LIN {X 0,Y 188.353,Z 512.177,A -85,B 0,C 180,E1 -22070.571,E2 -22070.571} C_VEL
LIN {X 0,Y 190.669,Z 502.352,A -85,B 0,C 180,E1 -22073.346,E2 -22073.346} C_VEL
LIN {X 0,Y 192.539,Z 493.281,A -85,B 0,C 180,E1 -22075.401,E2 -22075.401} C_VEL
LIN {X 0,Y 194.201,Z 485.139,A -85,B 0,C 180,E1 -22076.899,E2 -22076.899} C_VEL
LIN {X 0,Y 196.354,Z 473.565,A -85,B 0,C 180,E1 -22078.605,E2 -22078.605} C_VEL
LIN {X 0,Y 198.216,Z 461.568,A -85,B 0,C 180,E1 -22079.911,E2 -22079.911} C_VEL
LIN {X 0,Y 199.572,Z 449.492,A -85,B 0,C 180,E1 -22080.855,E2 -22080.855} C_VEL
LIN {X 0,Y 200.443,Z 436.398,A -85,B 0,C 180,E1 -22081.513,E2 -22081.513} C_VEL
LIN {X 0,Y 202.303,Z 391.383,A -85,B 0,C 180,E1 -22083.04,E2 -22083.04} C_VEL
LIN {X 0,Y 199.367,Z 363.798,A -85,B 0,C 180,E1 -22084.587,E2 -22084.587} C_VEL
LIN {X 0,Y 192.816,Z 346.528,A -85,B 0,C 180,E1 -22086.384,E2 -22086.384} C_VEL
LIN {X 0,Y 187.657,Z 334.98,A -85,B 0,C 180,E1 -22087.815,E2 -22087.815} C_VEL
LIN {X 0,Y 186.775,Z 332.616,A -85,B 0,C 180,E1 -22088.175,E2 -22088.175} C_VEL
LIN {X 0,Y 185.486,Z 327.382,A -85,B 0,C 180,E1 -22091.001,E2 -22091.001} C_VEL
LIN {X 0,Y 185.466,Z 327.381,A -85,B 0,C 180,E1 -22096.057,E2 -22096.057} C_VEL
LIN {X 0,Y 185.475,Z 327.377,A -85,B 0,C 180,E1 -22099.896,E2 -22099.896} C_VEL
LIN {X 0,Y 185.514,Z 327.371,A -85,B 0,C 180,E1 -22102.713,E2 -22102.713} C_VEL
LIN {X 0,Y 185.555,Z 327.368,A -85,B 0,C 180,E1 -22107.977,E2 -22107.977} C_VEL
LIN {X 0,Y 185.591,Z 327.36,A -85,B 0,C 180,E1 -22110.577,E2 -22110.577} C_VEL
LIN {X 0,Y 185.589,Z 327.367,A -85,B 0,C 180,E1 -22115.382,E2 -22115.382} C_VEL
LIN {X 0,Y 185.552,Z 327.357,A -85,B 0,C 180,E1 -22120.069,E2 -22120.069} C_VEL
LIN {X 0,Y 185.678,Z 327.348,A -85,B 0,C 180,E1 -22124.635,E2 -22124.635} C_VEL
LIN {X 0,Y 185.897,Z 327.323,A -85,B 0,C 180,E1 -22129.419,E2 -22129.419} C_VEL
LIN {X 0,Y 185.944,Z 327.291,A -85,B 0,C 180,E1 -22133.489,E2 -22133.489} C_VEL
LIN {X 0,Y 186.21,Z 327.284,A -85,B 0,C 180,E1 -22137.837,E2 -22137.837} C_VEL
LIN {X 0,Y 186.412,Z 327.264,A -85,B 0,C 180,E1 -22140,E2 -22140} C_VEL
LIN {X 0,Y 185.922,Z 327.297,A -85,B 0,C 180,E1 -22144.335,E2 -22144.335} C_VEL
LIN {X 0,Y 185.989,Z 327.3,A -85,B 0,C 180,E1 -22148.693,E2 -22148.693} C_VEL
LIN {X 0,Y 185.727,Z 327.348,A -85,B 0,C 180,E1 -22153.123,E2 -22153.123} C_VEL
LIN {X 0,Y 185.664,Z 327.355,A -85,B 0,C 180,E1 -22157.627,E2 -22157.627} C_VEL
LIN {X 0,Y 185.581,Z 327.36,A -85,B 0,C 180,E1 -22162.253,E2 -22162.253} C_VEL
LIN {X 0,Y 185.568,Z 327.366,A -85,B 0,C 180,E1 -22167.031,E2 -22167.031} C_VEL
LIN {X 0,Y 185.586,Z 327.36,A -85,B 0,C 180,E1 -22169.491,E2 -22169.491} C_VEL
LIN {X 0,Y 185.506,Z 327.367,A -85,B 0,C 180,E1 -22174.63,E2 -22174.63} C_VEL
LIN {X 0,Y 185.513,Z 327.374,A -85,B 0,C 180,E1 -22177.311,E2 -22177.311} C_VEL
LIN {X 0,Y 185.477,Z 327.37,A -85,B 0,C 180,E1 -22180.723,E2 -22180.723} C_VEL
LIN {X 0,Y 185.464,Z 327.376,A -85,B 0,C 180,E1 -22186.053,E2 -22186.053} C_VEL
LIN {X 0,Y 185.472,Z 327.376,A -85,B 0,C 180,E1 -22189.893,E2 -22189.893} C_VEL
LIN {X 0,Y 185.511,Z 327.376,A -85,B 0,C 180,E1 -22192.709,E2 -22192.709} C_VEL
LIN {X 0,Y 185.546,Z 327.37,A -85,B 0,C 180,E1 -22197.972,E2 -22197.972} C_VEL
LIN {X 0,Y 185.585,Z 327.368,A -85,B 0,C 180,E1 -22200.574,E2 -22200.574} C_VEL
LIN {X 0,Y 185.68,Z 327.355,A -85,B 0,C 180,E1 -22206.578,E2 -22206.578} C_VEL
LIN {X 0,Y 185.67,Z 327.485,A -85,B 0,C 180,E1 -22207.071,E2 -22207.071} C_VEL
LIN {X 0,Y 186.702,Z 330.28,A -85,B 0,C 180,E1 -22207.396,E2 -22207.396} C_VEL
LIN {X 0,Y 194.168,Z 343.936,A -85,B 0,C 180,E1 -22209.343,E2 -22209.343} C_VEL
LIN {X 0,Y 200.218,Z 357.134,A -85,B 0,C 180,E1 -22210.88,E2 -22210.88} C_VEL
LIN {X 0,Y 203.246,Z 366.009,A -85,B 0,C 180,E1 -22211.697,E2 -22211.697} C_VEL
LIN {X 0,Y 200.358,Z 428.689,A -85,B 0,C 180,E1 -22213.831,E2 -22213.831} C_VEL
LIN {X 0,Y 199.181,Z 442.535,A -85,B 0,C 180,E1 -22214.717,E2 -22214.717} C_VEL
LIN {X 0,Y 197.731,Z 455.437,A -85,B 0,C 180,E1 -22215.984,E2 -22215.984} C_VEL
LIN {X 0,Y 195.76,Z 467.279,A -85,B 0,C 180,E1 -22217.558,E2 -22217.558} C_VEL
LIN {X 0,Y 193.815,Z 478.594,A -85,B 0,C 180,E1 -22219.551,E2 -22219.551} C_VEL
LIN {X 0,Y 191.557,Z 488.867,A -85,B 0,C 180,E1 -22221.824,E2 -22221.824} C_VEL
LIN {X 0,Y 189.243,Z 498.9,A -85,B 0,C 180,E1 -22224.67,E2 -22224.67} C_VEL
LIN {X 0,Y 187.126,Z 507.738,A -85,B 0,C 180,E1 -22227.844,E2 -22227.844} C_VEL
LIN {X 0,Y 185.539,Z 514.774,A -85,B 0,C 180,E1 -22231.082,E2 -22231.082} C_VEL
LIN {X 0,Y 184.434,Z 520.402,A -85,B 0,C 180,E1 -22234.368,E2 -22234.368} C_VEL
LIN {X 0,Y 183.638,Z 524.836,A -85,B 0,C 180,E1 -22237.694,E2 -22237.694} C_VEL
LIN {X 0,Y 183.048,Z 528.196,A -85,B 0,C 180,E1 -22241.064,E2 -22241.064} C_VEL
LIN {X 0,Y 182.893,Z 529.868,A -85,B 0,C 180,E1 -22243.327,E2 -22243.327} C_VEL
LIN {X 0,Y 182.926,Z 531.341,A -85,B 0,C 180,E1 -22246.159,E2 -22246.159} C_VEL
LIN {X 0,Y 183.339,Z 532.303,A -85,B 0,C 180,E1 -22250.178,E2 -22250.178} C_VEL
LIN {X 0,Y 184.263,Z 532.066,A -85,B 0,C 180,E1 -22253.741,E2 -22253.741} C_VEL
LIN {X 0,Y 185.539,Z 530.916,A -85,B 0,C 180,E1 -22257.032,E2 -22257.032} C_VEL
LIN {X 0,Y 187.356,Z 528.771,A -85,B 0,C 180,E1 -22260.373,E2 -22260.373} C_VEL
LIN {X 0,Y 189.807,Z 525.491,A -85,B 0,C 180,E1 -22263.734,E2 -22263.734} C_VEL
LIN {X 0,Y 192.877,Z 520.967,A -85,B 0,C 180,E1 -22267.041,E2 -22267.041} C_VEL
LIN {X 0,Y 196.347,Z 515.364,A -85,B 0,C 180,E1 -22270.108,E2 -22270.108} C_VEL
LIN {X 0,Y 200.451,Z 508.123,A -85,B 0,C 180,E1 -22273.128,E2 -22273.128} C_VEL
LIN {X 0,Y 204.18,Z 500.616,A -85,B 0,C 180,E1 -22275.575,E2 -22275.575} C_VEL
LIN {X 0,Y 208.336,Z 491.441,A -85,B 0,C 180,E1 -22277.91,E2 -22277.91} C_VEL
LIN {X 0,Y 212.331,Z 481.267,A -85,B 0,C 180,E1 -22279.939,E2 -22279.939} C_VEL
LIN {X 0,Y 215.607,Z 471.5,A -85,B 0,C 180,E1 -22281.467,E2 -22281.467} C_VEL
LIN {X 0,Y 218.521,Z 460.893,A -85,B 0,C 180,E1 -22282.785,E2 -22282.785} C_VEL
LIN {X 0,Y 221.185,Z 448.606,A -85,B 0,C 180,E1 -22283.921,E2 -22283.921} C_VEL
LIN {X 0,Y 223.29,Z 435.152,A -85,B 0,C 180,E1 -22284.784,E2 -22284.784} C_VEL
LIN {X 0,Y 224.598,Z 421.235,A -85,B 0,C 180,E1 -22285.305,E2 -22285.305} C_VEL
LIN {X 0,Y 226.623,Z 388.171,A -85,B 0,C 180,E1 -22286.294,E2 -22286.294} C_VEL
LIN {X 0,Y 221.369,Z 377.129,A -85,B 0,C 180,E1 -22288.355,E2 -22288.355} C_VEL
LIN {X 0,Y 217.126,Z 369.65,A -85,B 0,C 180,E1 -22290.088,E2 -22290.088} C_VEL
LIN {X 0,Y 211.412,Z 360.897,A -85,B 0,C 180,E1 -22292.6,E2 -22292.6} C_VEL
LIN {X 0,Y 205.592,Z 352.678,A -85,B 0,C 180,E1 -22295.44,E2 -22295.44} C_VEL
LIN {X 0,Y 202.329,Z 348.373,A -85,B 0,C 180,E1 -22297.188,E2 -22297.188} C_VEL
LIN {X 0,Y 199.485,Z 344.709,A -85,B 0,C 180,E1 -22298.832,E2 -22298.832} C_VEL
LIN {X 0,Y 198.733,Z 343.71,A -85,B 0,C 180,E1 -22299.29,E2 -22299.29} C_VEL
LIN {X 0,Y 196.069,Z 340.766,A -85,B 0,C 180,E1 -22300.977,E2 -22300.977} C_VEL
LIN {X 0,Y 194.761,Z 338.596,A -85,B 0,C 180,E1 -22301.92,E2 -22301.92} C_VEL
LIN {X 0,Y 192.179,Z 336.315,A -85,B 0,C 180,E1 -22303.741,E2 -22303.741} C_VEL
LIN {X 0,Y 190.522,Z 333.195,A -85,B 0,C 180,E1 -22305.173,E2 -22305.173} C_VEL
LIN {X 0,Y 187.93,Z 331.617,A -85,B 0,C 180,E1 -22307.309,E2 -22307.309} C_VEL
LIN {X 0,Y 186.403,Z 329.386,A -85,B 0,C 180,E1 -22308.859,E2 -22308.859} C_VEL
LIN {X 0,Y 185.903,Z 327.319,A -85,B 0,C 180,E1 -22309.598,E2 -22309.598} C_VEL
LIN {X 0,Y 185.927,Z 327.307,A -85,B 0,C 180,E1 -22313.489,E2 -22313.489} C_VEL
LIN {X 0,Y 186.192,Z 327.272,A -85,B 0,C 180,E1 -22317.837,E2 -22317.837} C_VEL
LIN {X 0,Y 186.394,Z 327.258,A -85,B 0,C 180,E1 -22320,E2 -22320} C_VEL
LIN {X 0,Y 185.911,Z 327.309,A -85,B 0,C 180,E1 -22324.337,E2 -22324.337} C_VEL
LIN {X 0,Y 185.997,Z 327.295,A -85,B 0,C 180,E1 -22328.694,E2 -22328.694} C_VEL
LIN {X 0,Y 185.753,Z 327.328,A -85,B 0,C 180,E1 -22333.122,E2 -22333.122} C_VEL
LIN {X 0,Y 185.679,Z 327.343,A -85,B 0,C 180,E1 -22337.626,E2 -22337.626} C_VEL
LIN {X 0,Y 185.633,Z 327.508,A -85,B 0,C 180,E1 -22343.129,E2 -22343.129} C_VEL
LIN {X 0,Y 186.049,Z 329.192,A -85,B 0,C 180,E1 -22345.335,E2 -22345.335} C_VEL
LIN {X 0,Y 187.524,Z 331.42,A -85,B 0,C 180,E1 -22346.878,E2 -22346.878} C_VEL
LIN {X 0,Y 191.885,Z 336.607,A -85,B 0,C 180,E1 -22350.627,E2 -22350.627} C_VEL
LIN {X 0,Y 195.187,Z 341.306,A -85,B 0,C 180,E1 -22353.094,E2 -22353.094} C_VEL
LIN {X 0,Y 197.203,Z 343.952,A -85,B 0,C 180,E1 -22354.446,E2 -22354.446} C_VEL
LIN {X 0,Y 200.298,Z 348.364,A -85,B 0,C 180,E1 -22356.375,E2 -22356.375} C_VEL
LIN {X 0,Y 205.123,Z 355.887,A -85,B 0,C 180,E1 -22359.103,E2 -22359.103} C_VEL
LIN {X 0,Y 209.046,Z 362.3,A -85,B 0,C 180,E1 -22361.114,E2 -22361.114} C_VEL
LIN {X 0,Y 213.437,Z 369.913,A -85,B 0,C 180,E1 -22363.193,E2 -22363.193} C_VEL
LIN {X 0,Y 219.34,Z 381.612,A -85,B 0,C 180,E1 -22365.781,E2 -22365.781} C_VEL
LIN {X 0,Y 224.902,Z 394.525,A -85,B 0,C 180,E1 -22368.063,E2 -22368.063} C_VEL
LIN {X 0,Y 225.82,Z 397.48,A -85,B 0,C 180,E1 -22368.458,E2 -22368.458} C_VEL
LIN {X 0,Y 225.93,Z 401.219,A -85,B 0,C 180,E1 -22368.663,E2 -22368.663} C_VEL
LIN {X 0,Y 223.2,Z 441.55,A -85,B 0,C 180,E1 -22369.875,E2 -22369.875} C_VEL
LIN {X 0,Y 222.275,Z 449.228,A -85,B 0,C 180,E1 -22370.238,E2 -22370.238} C_VEL
LIN {X 0,Y 220.943,Z 454.939,A -85,B 0,C 180,E1 -22370.446,E2 -22370.446} C_VEL
LIN {X 0,Y 217.108,Z 464.094,A -85,B 0,C 180,E1 -22370.568,E2 -22370.568} C_VEL
LIN {X 0,Y 212.771,Z 472.95,A -85,B 0,C 180,E1 -22370.849,E2 -22370.849} C_VEL
LIN {X 0,Y 210.664,Z 478.188,A -85,B 0,C 180,E1 -22371.317,E2 -22371.317} C_VEL
LIN {X 0,Y 206.77,Z 489.566,A -85,B 0,C 180,E1 -22372.897,E2 -22372.897} C_VEL
LIN {X 0,Y 202.532,Z 499.986,A -85,B 0,C 180,E1 -22374.771,E2 -22374.771} C_VEL
LIN {X 0,Y 198.603,Z 508.522,A -85,B 0,C 180,E1 -22376.74,E2 -22376.74} C_VEL
LIN {X 0,Y 194.585,Z 516.413,A -85,B 0,C 180,E1 -22379.028,E2 -22379.028} C_VEL
LIN {X 0,Y 190.119,Z 524.183,A -85,B 0,C 180,E1 -22381.884,E2 -22381.884} C_VEL
LIN {X 0,Y 186.84,Z 529.738,A -85,B 0,C 180,E1 -22384.525,E2 -22384.525} C_VEL
LIN {X 0,Y 183.808,Z 534.686,A -85,B 0,C 180,E1 -22387.524,E2 -22387.524} C_VEL
LIN {X 0,Y 181.041,Z 538.753,A -85,B 0,C 180,E1 -22390.737,E2 -22390.737} C_VEL
LIN {X 0,Y 178.81,Z 541.797,A -85,B 0,C 180,E1 -22394.034,E2 -22394.034} C_VEL
LIN {X 0,Y 177.805,Z 543.321,A -85,B 0,C 180,E1 -22396.285,E2 -22396.285} C_VEL
LIN {X 0,Y 176.473,Z 545.123,A -85,B 0,C 180,E1 -22400.837,E2 -22400.837} C_VEL
LIN {X 0,Y 176.067,Z 545.411,A -85,B 0,C 180,E1 -22405.425,E2 -22405.425} C_VEL
LIN {X 0,Y 176.085,Z 544.94,A -85,B 0,C 180,E1 -22407.716,E2 -22407.716} C_VEL
LIN {X 0,Y 176.261,Z 544.069,A -85,B 0,C 180,E1 -22410.003,E2 -22410.003} C_VEL
LIN {X 0,Y 176.076,Z 541.728,A -85,B 0,C 180,E1 -22413.736,E2 -22413.736} C_VEL
LIN {X 0,Y 176.333,Z 537.6,A -85,B 0,C 180,E1 -22418.022,E2 -22418.022} C_VEL
LIN {X 0,Y 176.907,Z 533.014,A -85,B 0,C 180,E1 -22421.46,E2 -22421.46} C_VEL
LIN {X 0,Y 178.167,Z 526.023,A -85,B 0,C 180,E1 -22425.445,E2 -22425.445} C_VEL
LIN {X 0,Y 179.915,Z 518.437,A -85,B 0,C 180,E1 -22428.803,E2 -22428.803} C_VEL
LIN {X 0,Y 181.517,Z 511.685,A -85,B 0,C 180,E1 -22431.22,E2 -22431.22} C_VEL
LIN {X 0,Y 183.88,Z 502.268,A -85,B 0,C 180,E1 -22433.963,E2 -22433.963} C_VEL
LIN {X 0,Y 185.826,Z 493.232,A -85,B 0,C 180,E1 -22436.085,E2 -22436.085} C_VEL
LIN {X 0,Y 187.546,Z 485.126,A -85,B 0,C 180,E1 -22437.632,E2 -22437.632} C_VEL
LIN {X 0,Y 189.781,Z 473.623,A -85,B 0,C 180,E1 -22439.388,E2 -22439.388} C_VEL
LIN {X 0,Y 191.699,Z 461.749,A -85,B 0,C 180,E1 -22440.732,E2 -22440.732} C_VEL
LIN {X 0,Y 193.103,Z 449.847,A -85,B 0,C 180,E1 -22441.702,E2 -22441.702} C_VEL
LIN {X 0,Y 194.026,Z 437.151,A -85,B 0,C 180,E1 -22442.375,E2 -22442.375} C_VEL
LIN {X 0,Y 195.946,Z 391.813,A -85,B 0,C 180,E1 -22443.966,E2 -22443.966} C_VEL
LIN {X 0,Y 193.252,Z 365.907,A -85,B 0,C 180,E1 -22445.482,E2 -22445.482} C_VEL
LIN {X 0,Y 186.381,Z 347.697,A -85,B 0,C 180,E1 -22447.487,E2 -22447.487} C_VEL
LIN {X 0,Y 180.679,Z 335.314,A -85,B 0,C 180,E1 -22449.163,E2 -22449.163} C_VEL
LIN {X 0,Y 179.434,Z 332.329,A -85,B 0,C 180,E1 -22449.641,E2 -22449.641} C_VEL
LIN {X 0,Y 178.418,Z 328.26,A -85,B 0,C 180,E1 -22452.043,E2 -22452.043} C_VEL
LIN {X 0,Y 178.401,Z 328.264,A -85,B 0,C 180,E1 -22455.166,E2 -22455.166} C_VEL
LIN {X 0,Y 178.41,Z 328.26,A -85,B 0,C 180,E1 -22458.461,E2 -22458.461} C_VEL
LIN {X 0,Y 178.431,Z 328.255,A -85,B 0,C 180,E1 -22463.784,E2 -22463.784} C_VEL
LIN {X 0,Y 178.496,Z 328.244,A -85,B 0,C 180,E1 -22466.548,E2 -22466.548} C_VEL
LIN {X 0,Y 178.532,Z 328.238,A -85,B 0,C 180,E1 -22470.007,E2 -22470.007} C_VEL
LIN {X 0,Y 178.529,Z 328.247,A -85,B 0,C 180,E1 -22474.887,E2 -22474.887} C_VEL
LIN {X 0,Y 178.565,Z 328.219,A -85,B 0,C 180,E1 -22480.847,E2 -22480.847} C_VEL
LIN {X 0,Y 178.654,Z 328.229,A -85,B 0,C 180,E1 -22486.347,E2 -22486.347} C_VEL
LIN {X 0,Y 178.913,Z 328.181,A -85,B 0,C 180,E1 -22490.959,E2 -22490.959} C_VEL
LIN {X 0,Y 179.156,Z 328.162,A -85,B 0,C 180,E1 -22497.751,E2 -22497.751} C_VEL
LIN {X 0,Y 179.375,Z 328.14,A -85,B 0,C 180,E1 -22500,E2 -22500} C_VEL
LIN {X 0,Y 178.869,Z 328.173,A -85,B 0,C 180,E1 -22504.507,E2 -22504.507} C_VEL
LIN {X 0,Y 178.918,Z 328.183,A -85,B 0,C 180,E1 -22509.039,E2 -22509.039} C_VEL
LIN {X 0,Y 178.653,Z 328.228,A -85,B 0,C 180,E1 -22513.652,E2 -22513.652} C_VEL
LIN {X 0,Y 178.598,Z 328.238,A -85,B 0,C 180,E1 -22519.184,E2 -22519.184} C_VEL
LIN {X 0,Y 178.528,Z 328.247,A -85,B 0,C 180,E1 -22525.113,E2 -22525.113} C_VEL
LIN {X 0,Y 178.53,Z 328.24,A -85,B 0,C 180,E1 -22529.992,E2 -22529.992} C_VEL
LIN {X 0,Y 178.492,Z 328.242,A -85,B 0,C 180,E1 -22534.217,E2 -22534.217} C_VEL
LIN {X 0,Y 178.402,Z 328.256,A -85,B 0,C 180,E1 -22539.072,E2 -22539.072} C_VEL
LIN {X 0,Y 178.404,Z 328.258,A -85,B 0,C 180,E1 -22542.043,E2 -22542.043} C_VEL
LIN {X 0,Y 178.399,Z 328.255,A -85,B 0,C 180,E1 -22545.162,E2 -22545.162} C_VEL
LIN {X 0,Y 178.408,Z 328.259,A -85,B 0,C 180,E1 -22548.457,E2 -22548.457} C_VEL
LIN {X 0,Y 178.427,Z 328.256,A -85,B 0,C 180,E1 -22553.781,E2 -22553.781} C_VEL
LIN {X 0,Y 178.49,Z 328.252,A -85,B 0,C 180,E1 -22556.544,E2 -22556.544} C_VEL
LIN {X 0,Y 178.526,Z 328.248,A -85,B 0,C 180,E1 -22560.004,E2 -22560.004} C_VEL
LIN {X 0,Y 178.594,Z 328.324,A -85,B 0,C 180,E1 -22565.674,E2 -22565.674} C_VEL
LIN {X 0,Y 179.692,Z 331.231,A -85,B 0,C 180,E1 -22566.044,E2 -22566.044} C_VEL
LIN {X 0,Y 180.979,Z 333.249,A -85,B 0,C 180,E1 -22566.404,E2 -22566.404} C_VEL
LIN {X 0,Y 189.443,Z 349.04,A -85,B 0,C 180,E1 -22568.736,E2 -22568.736} C_VEL
LIN {X 0,Y 194.932,Z 361.55,A -85,B 0,C 180,E1 -22570.217,E2 -22570.217} C_VEL
LIN {X 0,Y 196.911,Z 367.636,A -85,B 0,C 180,E1 -22570.79,E2 -22570.79} C_VEL
LIN {X 0,Y 193.961,Z 429.467,A -85,B 0,C 180,E1 -22572.966,E2 -22572.966} C_VEL
LIN {X 0,Y 192.748,Z 442.893,A -85,B 0,C 180,E1 -22573.855,E2 -22573.855} C_VEL
LIN {X 0,Y 191.305,Z 455.251,A -85,B 0,C 180,E1 -22575.095,E2 -22575.095} C_VEL
LIN {X 0,Y 189.392,Z 466.403,A -85,B 0,C 180,E1 -22576.586,E2 -22576.586} C_VEL
LIN {X 0,Y 187.311,Z 477.935,A -85,B 0,C 180,E1 -22578.636,E2 -22578.636} C_VEL
LIN {X 0,Y 185.047,Z 488.117,A -85,B 0,C 180,E1 -22580.917,E2 -22580.917} C_VEL
LIN {X 0,Y 182.954,Z 496.91,A -85,B 0,C 180,E1 -22583.379,E2 -22583.379} C_VEL
LIN {X 0,Y 180.629,Z 506.146,A -85,B 0,C 180,E1 -22586.651,E2 -22586.651} C_VEL
LIN {X 0,Y 178.833,Z 513.573,A -85,B 0,C 180,E1 -22589.997,E2 -22589.997} C_VEL
LIN {X 0,Y 177.587,Z 519.52,A -85,B 0,C 180,E1 -22593.4,E2 -22593.4} C_VEL
LIN {X 0,Y 176.719,Z 524.218,A -85,B 0,C 180,E1 -22596.849,E2 -22596.849} C_VEL
LIN {X 0,Y 176.048,Z 527.816,A -85,B 0,C 180,E1 -22600.345,E2 -22600.345} C_VEL
LIN {X 0,Y 175.805,Z 530.377,A -85,B 0,C 180,E1 -22603.874,E2 -22603.874} C_VEL
LIN {X 0,Y 175.841,Z 531.6,A -85,B 0,C 180,E1 -22606.418,E2 -22606.418} C_VEL
LIN {X 0,Y 176.038,Z 532.27,A -85,B 0,C 180,E1 -22608.622,E2 -22608.622} C_VEL
LIN {X 0,Y 176.387,Z 532.605,A -85,B 0,C 180,E1 -22611.01,E2 -22611.01} C_VEL
LIN {X 0,Y 177.311,Z 532.347,A -85,B 0,C 180,E1 -22614.268,E2 -22614.268} C_VEL
LIN {X 0,Y 178.897,Z 531.002,A -85,B 0,C 180,E1 -22618.122,E2 -22618.122} C_VEL
LIN {X 0,Y 180.653,Z 529.082,A -85,B 0,C 180,E1 -22621.145,E2 -22621.145} C_VEL
LIN {X 0,Y 183.609,Z 525.347,A -85,B 0,C 180,E1 -22625.036,E2 -22625.036} C_VEL
LIN {X 0,Y 186.754,Z 520.975,A -85,B 0,C 180,E1 -22628.242,E2 -22628.242} C_VEL
LIN {X 0,Y 190.672,Z 514.949,A -85,B 0,C 180,E1 -22631.56,E2 -22631.56} C_VEL
LIN {X 0,Y 195.041,Z 507.482,A -85,B 0,C 180,E1 -22634.635,E2 -22634.635} C_VEL
LIN {X 0,Y 199.026,Z 499.801,A -85,B 0,C 180,E1 -22637.11,E2 -22637.11} C_VEL
LIN {X 0,Y 203.443,Z 490.423,A -85,B 0,C 180,E1 -22639.458,E2 -22639.458} C_VEL
LIN {X 0,Y 207.631,Z 479.918,A -85,B 0,C 180,E1 -22641.507,E2 -22641.507} C_VEL
LIN {X 0,Y 211.037,Z 469.743,A -85,B 0,C 180,E1 -22643.053,E2 -22643.053} C_VEL
LIN {X 0,Y 214.219,Z 458.058,A -85,B 0,C 180,E1 -22644.426,E2 -22644.426} C_VEL
LIN {X 0,Y 216.844,Z 445.648,A -85,B 0,C 180,E1 -22645.497,E2 -22645.497} C_VEL
LIN {X 0,Y 218.807,Z 432.093,A -85,B 0,C 180,E1 -22646.272,E2 -22646.272} C_VEL
LIN {X 0,Y 220.443,Z 411.955,A -85,B 0,C 180,E1 -22646.911,E2 -22646.911} C_VEL
LIN {X 0,Y 221.806,Z 390.87,A -85,B 0,C 180,E1 -22647.543,E2 -22647.543} C_VEL
LIN {X 0,Y 215.986,Z 378.812,A -85,B 0,C 180,E1 -22649.981,E2 -22649.981} C_VEL
LIN {X 0,Y 210.766,Z 370.185,A -85,B 0,C 180,E1 -22652.307,E2 -22652.307} C_VEL
LIN {X 0,Y 205.049,Z 361.765,A -85,B 0,C 180,E1 -22655.095,E2 -22655.095} C_VEL
LIN {X 0,Y 201.995,Z 357.486,A -85,B 0,C 180,E1 -22656.727,E2 -22656.727} C_VEL
LIN {X 0,Y 199.787,Z 354.448,A -85,B 0,C 180,E1 -22657.985,E2 -22657.985} C_VEL
LIN {X 0,Y 196.313,Z 349.896,A -85,B 0,C 180,E1 -22660.118,E2 -22660.118} C_VEL
LIN {X 0,Y 193.576,Z 346.506,A -85,B 0,C 180,E1 -22661.97,E2 -22661.97} C_VEL
LIN {X 0,Y 192.732,Z 345.096,A -85,B 0,C 180,E1 -22662.608,E2 -22662.608} C_VEL
LIN {X 0,Y 190.063,Z 342.457,A -85,B 0,C 180,E1 -22664.613,E2 -22664.613} C_VEL
LIN {X 0,Y 188.536,Z 339.837,A -85,B 0,C 180,E1 -22665.978,E2 -22665.978} C_VEL
LIN {X 0,Y 186.034,Z 337.952,A -85,B 0,C 180,E1 -22668.192,E2 -22668.192} C_VEL
LIN {X 0,Y 184.445,Z 335.196,A -85,B 0,C 180,E1 -22669.97,E2 -22669.97} C_VEL
LIN {X 0,Y 184.082,Z 334.182,A -85,B 0,C 180,E1 -22670.458,E2 -22670.458} C_VEL
LIN {X 0,Y 180.865,Z 332.321,A -85,B 0,C 180,E1 -22674.426,E2 -22674.426} C_VEL
LIN {X 0,Y 179.588,Z 330.34,A -85,B 0,C 180,E1 -22676.705,E2 -22676.705} C_VEL
LIN {X 0,Y 179.174,Z 328.146,A -85,B 0,C 180,E1 -22678.034,E2 -22678.034} C_VEL
LIN {X 0,Y 179.357,Z 328.134,A -85,B 0,C 180,E1 -22680,E2 -22680} C_VEL
LIN {X 0,Y 178.859,Z 328.188,A -85,B 0,C 180,E1 -22684.508,E2 -22684.508} C_VEL
LIN {X 0,Y 178.927,Z 328.176,A -85,B 0,C 180,E1 -22689.04,E2 -22689.04} C_VEL
LIN {X 0,Y 178.657,Z 328.214,A -85,B 0,C 180,E1 -22694.815,E2 -22694.815} C_VEL
LIN {X 0,Y 178.684,Z 328.396,A -85,B 0,C 180,E1 -22695.689,E2 -22695.689} C_VEL
LIN {X 0,Y 179.242,Z 330.368,A -85,B 0,C 180,E1 -22697.249,E2 -22697.249} C_VEL
LIN {X 0,Y 181.445,Z 333.144,A -85,B 0,C 180,E1 -22700.995,E2 -22700.995} C_VEL
LIN {X 0,Y 183.191,Z 334.322,A -85,B 0,C 180,E1 -22703.179,E2 -22703.179} C_VEL
LIN {X 0,Y 184.599,Z 336.121,A -85,B 0,C 180,E1 -22704.833,E2 -22704.833} C_VEL
LIN {X 0,Y 189.954,Z 343.068,A -85,B 0,C 180,E1 -22709.911,E2 -22709.911} C_VEL
LIN {X 0,Y 193.654,Z 348.334,A -85,B 0,C 180,E1 -22712.768,E2 -22712.768} C_VEL
LIN {X 0,Y 195.185,Z 350.653,A -85,B 0,C 180,E1 -22713.85,E2 -22713.85} C_VEL
LIN {X 0,Y 198.605,Z 355.726,A -85,B 0,C 180,E1 -22716.058,E2 -22716.058} C_VEL
LIN {X 0,Y 202.34,Z 361.704,A -85,B 0,C 180,E1 -22718.251,E2 -22718.251} C_VEL
LIN {X 0,Y 207.433,Z 370.205,A -85,B 0,C 180,E1 -22720.949,E2 -22720.949} C_VEL
LIN {X 0,Y 212.701,Z 380.436,A -85,B 0,C 180,E1 -22723.516,E2 -22723.516} C_VEL
LIN {X 0,Y 217.233,Z 390.26,A -85,B 0,C 180,E1 -22725.56,E2 -22725.56} C_VEL
LIN {X 0,Y 221.015,Z 399.593,A -85,B 0,C 180,E1 -22727.188,E2 -22727.188} C_VEL
LIN {X 0,Y 221.116,Z 401.913,A -85,B 0,C 180,E1 -22727.331,E2 -22727.331} C_VEL
LIN {X 0,Y 218.279,Z 441.898,A -85,B 0,C 180,E1 -22728.555,E2 -22728.555} C_VEL
LIN {X 0,Y 216.296,Z 455.361,A -85,B 0,C 180,E1 -22729.258,E2 -22729.258} C_VEL
LIN {X 0,Y 213.624,Z 467.911,A -85,B 0,C 180,E1 -22730.252,E2 -22730.252} C_VEL
LIN {X 0,Y 210.664,Z 478.188,A -85,B 0,C 180,E1 -22731.317,E2 -22731.317} C_VEL
LIN {X 0,Y 208.463,Z 483.41,A -85,B 0,C 180,E1 -22731.858,E2 -22731.858} C_VEL
LIN {X 0,Y 203.377,Z 491.567,A -85,B 0,C 180,E1 -22732.555,E2 -22732.555} C_VEL
LIN {X 0,Y 198.034,Z 499.212,A -85,B 0,C 180,E1 -22733.434,E2 -22733.434} C_VEL
LIN {X 0,Y 195.439,Z 503.608,A -85,B 0,C 180,E1 -22734.261,E2 -22734.261} C_VEL
LIN {X 0,Y 191.046,Z 512.275,A -85,B 0,C 180,E1 -22736.513,E2 -22736.513} C_VEL
LIN {X 0,Y 186.159,Z 520.789,A -85,B 0,C 180,E1 -22739.363,E2 -22739.363} C_VEL
LIN {X 0,Y 181.833,Z 527.634,A -85,B 0,C 180,E1 -22742.371,E2 -22742.371} C_VEL
LIN {X 0,Y 178.381,Z 533.14,A -85,B 0,C 180,E1 -22745.567,E2 -22745.567} C_VEL
LIN {X 0,Y 175.255,Z 537.494,A -85,B 0,C 180,E1 -22748.848,E2 -22748.848} C_VEL
LIN {X 0,Y 173.469,Z 539.814,A -85,B 0,C 180,E1 -22751.092,E2 -22751.092} C_VEL
LIN {X 0,Y 171.967,Z 541.716,A -85,B 0,C 180,E1 -22753.381,E2 -22753.381} C_VEL
LIN {X 0,Y 170.057,Z 544.23,A -85,B 0,C 180,E1 -22758.078,E2 -22758.078} C_VEL
LIN {X 0,Y 169.093,Z 545.207,A -85,B 0,C 180,E1 -22762.841,E2 -22762.841} C_VEL
LIN {X 0,Y 169.002,Z 544.893,A -85,B 0,C 180,E1 -22766.428,E2 -22766.428} C_VEL
LIN {X 0,Y 169.18,Z 543.687,A -85,B 0,C 180,E1 -22770.004,E2 -22770.004} C_VEL
LIN {X 0,Y 169.003,Z 541.513,A -85,B 0,C 180,E1 -22773.579,E2 -22773.579} C_VEL
LIN {X 0,Y 169.157,Z 538.331,A -85,B 0,C 180,E1 -22777.164,E2 -22777.164} C_VEL
LIN {X 0,Y 169.654,Z 534.05,A -85,B 0,C 180,E1 -22780.747,E2 -22780.747} C_VEL
LIN {X 0,Y 170.793,Z 527.523,A -85,B 0,C 180,E1 -22784.906,E2 -22784.906} C_VEL
LIN {X 0,Y 172.524,Z 520.355,A -85,B 0,C 180,E1 -22788.407,E2 -22788.407} C_VEL
LIN {X 0,Y 174.385,Z 513.038,A -85,B 0,C 180,E1 -22791.27,E2 -22791.27} C_VEL
LIN {X 0,Y 175.788,Z 507.141,A -85,B 0,C 180,E1 -22793.207,E2 -22793.207} C_VEL
LIN {X 0,Y 177.781,Z 498.949,A -85,B 0,C 180,E1 -22795.465,E2 -22795.465} C_VEL
LIN {X 0,Y 180.219,Z 487.954,A -85,B 0,C 180,E1 -22797.906,E2 -22797.906} C_VEL
LIN {X 0,Y 182.599,Z 477.237,A -85,B 0,C 180,E1 -22799.709,E2 -22799.709} C_VEL
LIN {X 0,Y 184.666,Z 465.417,A -85,B 0,C 180,E1 -22801.238,E2 -22801.238} C_VEL
LIN {X 0,Y 186.369,Z 452.737,A -85,B 0,C 180,E1 -22802.428,E2 -22802.428} C_VEL
LIN {X 0,Y 187.599,Z 439.418,A -85,B 0,C 180,E1 -22803.226,E2 -22803.226} C_VEL
LIN {X 0,Y 189.692,Z 393.126,A -85,B 0,C 180,E1 -22804.909,E2 -22804.909} C_VEL
LIN {X 0,Y 187.213,Z 367.905,A -85,B 0,C 180,E1 -22806.435,E2 -22806.435} C_VEL
LIN {X 0,Y 180.304,Z 349.879,A -85,B 0,C 180,E1 -22808.558,E2 -22808.558} C_VEL
LIN {X 0,Y 174.117,Z 336.318,A -85,B 0,C 180,E1 -22810.516,E2 -22810.516} C_VEL
LIN {X 0,Y 172.072,Z 332.04,A -85,B 0,C 180,E1 -22811.261,E2 -22811.261} C_VEL
LIN {X 0,Y 171.331,Z 329.145,A -85,B 0,C 180,E1 -22813.093,E2 -22813.093} C_VEL
LIN {X 0,Y 171.343,Z 329.141,A -85,B 0,C 180,E1 -22817.592,E2 -22817.592} C_VEL
LIN {X 0,Y 171.395,Z 329.13,A -85,B 0,C 180,E1 -22822.042,E2 -22822.042} C_VEL
LIN {X 0,Y 171.407,Z 329.128,A -85,B 0,C 180,E1 -22825.094,E2 -22825.094} C_VEL
LIN {X 0,Y 171.458,Z 329.12,A -85,B 0,C 180,E1 -22830.535,E2 -22830.535} C_VEL
LIN {X 0,Y 171.452,Z 329.128,A -85,B 0,C 180,E1 -22835.8,E2 -22835.8} C_VEL
LIN {X 0,Y 171.519,Z 329.095,A -85,B 0,C 180,E1 -22840.864,E2 -22840.864} C_VEL
LIN {X 0,Y 171.568,Z 329.11,A -85,B 0,C 180,E1 -22845.772,E2 -22845.772} C_VEL
LIN {X 0,Y 171.852,Z 329.064,A -85,B 0,C 180,E1 -22850.585,E2 -22850.585} C_VEL
LIN {X 0,Y 171.812,Z 329.061,A -85,B 0,C 180,E1 -22855.307,E2 -22855.307} C_VEL
LIN {X 0,Y 172.339,Z 329.016,A -85,B 0,C 180,E1 -22859.999,E2 -22859.999} C_VEL
LIN {X 0,Y 171.817,Z 329.048,A -85,B 0,C 180,E1 -22864.692,E2 -22864.692} C_VEL
LIN {X 0,Y 171.855,Z 329.066,A -85,B 0,C 180,E1 -22869.414,E2 -22869.414} C_VEL
LIN {X 0,Y 171.567,Z 329.109,A -85,B 0,C 180,E1 -22874.227,E2 -22874.227} C_VEL
LIN {X 0,Y 171.523,Z 329.118,A -85,B 0,C 180,E1 -22879.532,E2 -22879.532} C_VEL
LIN {X 0,Y 171.467,Z 329.125,A -85,B 0,C 180,E1 -22885.607,E2 -22885.607} C_VEL
LIN {X 0,Y 171.449,Z 329.122,A -85,B 0,C 180,E1 -22890.585,E2 -22890.585} C_VEL
LIN {X 0,Y 171.4,Z 329.123,A -85,B 0,C 180,E1 -22895.033,E2 -22895.033} C_VEL
LIN {X 0,Y 171.364,Z 329.135,A -85,B 0,C 180,E1 -22898.805,E2 -22898.805} C_VEL
LIN {X 0,Y 171.326,Z 329.138,A -85,B 0,C 180,E1 -22904.215,E2 -22904.215} C_VEL
LIN {X 0,Y 171.34,Z 329.139,A -85,B 0,C 180,E1 -22908.979,E2 -22908.979} C_VEL
LIN {X 0,Y 171.392,Z 329.135,A -85,B 0,C 180,E1 -22912.038,E2 -22912.038} C_VEL
LIN {X 0,Y 171.403,Z 329.129,A -85,B 0,C 180,E1 -22915.09,E2 -22915.09} C_VEL
LIN {X 0,Y 171.452,Z 329.128,A -85,B 0,C 180,E1 -22920.531,E2 -22920.531} C_VEL
LIN {X 0,Y 171.487,Z 329.289,A -85,B 0,C 180,E1 -22924.136,E2 -22924.136} C_VEL
LIN {X 0,Y 172.559,Z 332.049,A -85,B 0,C 180,E1 -22924.525,E2 -22924.525} C_VEL
LIN {X 0,Y 174.052,Z 334.244,A -85,B 0,C 180,E1 -22924.972,E2 -22924.972} C_VEL
LIN {X 0,Y 182.286,Z 349.283,A -85,B 0,C 180,E1 -22927.411,E2 -22927.411} C_VEL
LIN {X 0,Y 188.468,Z 362.642,A -85,B 0,C 180,E1 -22929.16,E2 -22929.16} C_VEL
LIN {X 0,Y 190.604,Z 368.823,A -85,B 0,C 180,E1 -22929.801,E2 -22929.801} C_VEL
LIN {X 0,Y 187.659,Z 429.43,A -85,B 0,C 180,E1 -22931.996,E2 -22931.996} C_VEL
LIN {X 0,Y 186.435,Z 442.497,A -85,B 0,C 180,E1 -22932.869,E2 -22932.869} C_VEL
LIN {X 0,Y 184.942,Z 455.032,A -85,B 0,C 180,E1 -22934.146,E2 -22934.146} C_VEL
LIN {X 0,Y 182.774,Z 467.116,A -85,B 0,C 180,E1 -22935.807,E2 -22935.807} C_VEL
LIN {X 0,Y 180.613,Z 478.563,A -85,B 0,C 180,E1 -22937.924,E2 -22937.924} C_VEL
LIN {X 0,Y 178.261,Z 488.657,A -85,B 0,C 180,E1 -22940.274,E2 -22940.274} C_VEL
LIN {X 0,Y 175.868,Z 498.246,A -85,B 0,C 180,E1 -22943.111,E2 -22943.111} C_VEL
LIN {X 0,Y 173.511,Z 507.284,A -85,B 0,C 180,E1 -22946.513,E2 -22946.513} C_VEL
LIN {X 0,Y 171.678,Z 514.559,A -85,B 0,C 180,E1 -22949.997,E2 -22949.997} C_VEL
LIN {X 0,Y 170.424,Z 520.345,A -85,B 0,C 180,E1 -22953.543,E2 -22953.543} C_VEL
LIN {X 0,Y 169.558,Z 524.908,A -85,B 0,C 180,E1 -22957.139,E2 -22957.139} C_VEL
LIN {X 0,Y 169.062,Z 527.335,A -85,B 0,C 180,E1 -22959.568,E2 -22959.568} C_VEL
LIN {X 0,Y 168.751,Z 529.326,A -85,B 0,C 180,E1 -22962.015,E2 -22962.015} C_VEL
LIN {X 0,Y 168.691,Z 530.861,A -85,B 0,C 180,E1 -22964.472,E2 -22964.472} C_VEL
LIN {X 0,Y 168.773,Z 531.943,A -85,B 0,C 180,E1 -22966.943,E2 -22966.943} C_VEL
LIN {X 0,Y 169.034,Z 532.625,A -85,B 0,C 180,E1 -22969.424,E2 -22969.424} C_VEL
LIN {X 0,Y 169.494,Z 532.902,A -85,B 0,C 180,E1 -22971.908,E2 -22971.908} C_VEL
LIN {X 0,Y 170.388,Z 532.625,A -85,B 0,C 180,E1 -22974.848,E2 -22974.848} C_VEL
LIN {X 0,Y 172.324,Z 531.089,A -85,B 0,C 180,E1 -22979.297,E2 -22979.297} C_VEL
LIN {X 0,Y 173.966,Z 529.403,A -85,B 0,C 180,E1 -22981.966,E2 -22981.966} C_VEL
LIN {X 0,Y 176.496,Z 526.482,A -85,B 0,C 180,E1 -22985.262,E2 -22985.262} C_VEL
LIN {X 0,Y 179.813,Z 522.212,A -85,B 0,C 180,E1 -22988.704,E2 -22988.704} C_VEL
LIN {X 0,Y 183.729,Z 516.654,A -85,B 0,C 180,E1 -22992.017,E2 -22992.017} C_VEL
LIN {X 0,Y 188.207,Z 509.617,A -85,B 0,C 180,E1 -22995.189,E2 -22995.189} C_VEL
LIN {X 0,Y 192.275,Z 502.349,A -85,B 0,C 180,E1 -22997.741,E2 -22997.741} C_VEL
LIN {X 0,Y 196.967,Z 493.038,A -85,B 0,C 180,E1 -23000.263,E2 -23000.263} C_VEL
LIN {X 0,Y 201.57,Z 482.391,A -85,B 0,C 180,E1 -23002.48,E2 -23002.48} C_VEL
LIN {X 0,Y 205.586,Z 471.369,A -85,B 0,C 180,E1 -23004.243,E2 -23004.243} C_VEL
LIN {X 0,Y 208.986,Z 459.559,A -85,B 0,C 180,E1 -23005.685,E2 -23005.685} C_VEL
LIN {X 0,Y 211.917,Z 446.536,A -85,B 0,C 180,E1 -23006.838,E2 -23006.838} C_VEL
LIN {X 0,Y 213.863,Z 434.037,A -85,B 0,C 180,E1 -23007.596,E2 -23007.596} C_VEL
LIN {X 0,Y 215.294,Z 418.18,A -85,B 0,C 180,E1 -23008.15,E2 -23008.15} C_VEL
LIN {X 0,Y 216.928,Z 393.338,A -85,B 0,C 180,E1 -23008.913,E2 -23008.913} C_VEL
LIN {X 0,Y 211.965,Z 382.995,A -85,B 0,C 180,E1 -23011.141,E2 -23011.141} C_VEL
LIN {X 0,Y 207.033,Z 374.759,A -85,B 0,C 180,E1 -23013.474,E2 -23013.474} C_VEL
LIN {X 0,Y 200.537,Z 364.899,A -85,B 0,C 180,E1 -23016.902,E2 -23016.902} C_VEL
LIN {X 0,Y 197.015,Z 360.199,A -85,B 0,C 180,E1 -23018.964,E2 -23018.964} C_VEL
LIN {X 0,Y 194.123,Z 356.21,A -85,B 0,C 180,E1 -23020.847,E2 -23020.847} C_VEL
LIN {X 0,Y 191.255,Z 352.435,A -85,B 0,C 180,E1 -23022.904,E2 -23022.904} C_VEL
LIN {X 0,Y 190.317,Z 351.273,A -85,B 0,C 180,E1 -23023.623,E2 -23023.623} C_VEL
LIN {X 0,Y 187.66,Z 348.029,A -85,B 0,C 180,E1 -23025.812,E2 -23025.812} C_VEL
LIN {X 0,Y 186.752,Z 346.503,A -85,B 0,C 180,E1 -23026.669,E2 -23026.669} C_VEL
LIN {X 0,Y 184.158,Z 344.201,A -85,B 0,C 180,E1 -23029.126,E2 -23029.126} C_VEL
LIN {X 0,Y 182.523,Z 341.01,A -85,B 0,C 180,E1 -23031.141,E2 -23031.141} C_VEL
LIN {X 0,Y 179.44,Z 338.95,A -85,B 0,C 180,E1 -23035.226,E2 -23035.226} C_VEL
LIN {X 0,Y 178.274,Z 336.704,A -85,B 0,C 180,E1 -23037.6,E2 -23037.6} C_VEL
LIN {X 0,Y 177.833,Z 335.104,A -85,B 0,C 180,E1 -23038.868,E2 -23038.868} C_VEL
LIN {X 0,Y 176.021,Z 334.663,A -85,B 0,C 180,E1 -23049.19,E2 -23049.19} C_VEL
LIN {X 0,Y 177.53,Z 335.301,A -85,B 0,C 180,E1 -23055.058,E2 -23055.058} C_VEL
LIN {X 0,Y 178.496,Z 337.947,A -85,B 0,C 180,E1 -23057.619,E2 -23057.619} C_VEL
LIN {X 0,Y 180.706,Z 340.354,A -85,B 0,C 180,E1 -23061.234,E2 -23061.234} C_VEL
LIN {X 0,Y 182.063,Z 341.354,A -85,B 0,C 180,E1 -23062.952,E2 -23062.952} C_VEL
LIN {X 0,Y 183.135,Z 342.91,A -85,B 0,C 180,E1 -23064.277,E2 -23064.277} C_VEL
LIN {X 0,Y 188.048,Z 349.515,A -85,B 0,C 180,E1 -23069.167,E2 -23069.167} C_VEL
LIN {X 0,Y 192.554,Z 356.145,A -85,B 0,C 180,E1 -23072.762,E2 -23072.762} C_VEL
LIN {X 0,Y 196.082,Z 361.659,A -85,B 0,C 180,E1 -23075.195,E2 -23075.195} C_VEL
LIN {X 0,Y 199.721,Z 367.758,A -85,B 0,C 180,E1 -23077.449,E2 -23077.449} C_VEL
LIN {X 0,Y 203.726,Z 374.647,A -85,B 0,C 180,E1 -23079.698,E2 -23079.698} C_VEL
LIN {X 0,Y 208.364,Z 383.601,A -85,B 0,C 180,E1 -23082.107,E2 -23082.107} C_VEL
LIN {X 0,Y 213.002,Z 393.917,A -85,B 0,C 180,E1 -23084.362,E2 -23084.362} C_VEL
LIN {X 0,Y 216.392,Z 402.35,A -85,B 0,C 180,E1 -23085.917,E2 -23085.917} C_VEL
LIN {X 0,Y 213.631,Z 441.035,A -85,B 0,C 180,E1 -23087.124,E2 -23087.124} C_VEL
LIN {X 0,Y 211.536,Z 455.038,A -85,B 0,C 180,E1 -23087.857,E2 -23087.857} C_VEL
LIN {X 0,Y 208.797,Z 467.376,A -85,B 0,C 180,E1 -23088.822,E2 -23088.822} C_VEL
LIN {X 0,Y 205.271,Z 479.105,A -85,B 0,C 180,E1 -23090.067,E2 -23090.067} C_VEL
LIN {X 0,Y 201.178,Z 490.411,A -85,B 0,C 180,E1 -23091.682,E2 -23091.682} C_VEL
LIN {X 0,Y 196.806,Z 500.638,A -85,B 0,C 180,E1 -23093.585,E2 -23093.585} C_VEL
LIN {X 0,Y 195.439,Z 503.608,A -85,B 0,C 180,E1 -23094.261,E2 -23094.261} C_VEL
LIN {X 0,Y 192.768,Z 507.914,A -85,B 0,C 180,E1 -23095.175,E2 -23095.175} C_VEL
LIN {X 0,Y 186.934,Z 514.544,A -85,B 0,C 180,E1 -23096.536,E2 -23096.536} C_VEL
LIN {X 0,Y 180.997,Z 520.587,A -85,B 0,C 180,E1 -23098.132,E2 -23098.132} C_VEL
LIN {X 0,Y 178.217,Z 523.91,A -85,B 0,C 180,E1 -23099.409,E2 -23099.409} C_VEL
LIN {X 0,Y 174.275,Z 529.761,A -85,B 0,C 180,E1 -23102.375,E2 -23102.375} C_VEL
LIN {X 0,Y 170.764,Z 534.778,A -85,B 0,C 180,E1 -23105.701,E2 -23105.701} C_VEL
LIN {X 0,Y 167.684,Z 538.699,A -85,B 0,C 180,E1 -23109.134,E2 -23109.134} C_VEL
LIN {X 0,Y 165.155,Z 541.621,A -85,B 0,C 180,E1 -23112.674,E2 -23112.674} C_VEL
LIN {X 0,Y 163.098,Z 544.047,A -85,B 0,C 180,E1 -23117.562,E2 -23117.562} C_VEL
LIN {X 0,Y 162.023,Z 544.952,A -85,B 0,C 180,E1 -23122.527,E2 -23122.527} C_VEL
LIN {X 0,Y 161.913,Z 544.487,A -85,B 0,C 180,E1 -23126.706,E2 -23126.706} C_VEL
LIN {X 0,Y 162.082,Z 543.305,A -85,B 0,C 180,E1 -23130.004,E2 -23130.004} C_VEL
LIN {X 0,Y 161.914,Z 541.372,A -85,B 0,C 180,E1 -23133.301,E2 -23133.301} C_VEL
LIN {X 0,Y 162.113,Z 537.806,A -85,B 0,C 180,E1 -23137.477,E2 -23137.477} C_VEL
LIN {X 0,Y 162.642,Z 533.445,A -85,B 0,C 180,E1 -23141.216,E2 -23141.216} C_VEL
LIN {X 0,Y 163.638,Z 527.853,A -85,B 0,C 180,E1 -23144.937,E2 -23144.937} C_VEL
LIN {X 0,Y 165.425,Z 520.873,A -85,B 0,C 180,E1 -23148.584,E2 -23148.584} C_VEL
LIN {X 0,Y 167.643,Z 512.072,A -85,B 0,C 180,E1 -23152.17,E2 -23152.17} C_VEL
LIN {X 0,Y 170.371,Z 502.07,A -85,B 0,C 180,E1 -23155.343,E2 -23155.343} C_VEL
LIN {X 0,Y 172.491,Z 493.103,A -85,B 0,C 180,E1 -23157.615,E2 -23157.615} C_VEL
LIN {X 0,Y 174.34,Z 485.077,A -85,B 0,C 180,E1 -23159.264,E2 -23159.264} C_VEL
LIN {X 0,Y 176.738,Z 473.689,A -85,B 0,C 180,E1 -23161.131,E2 -23161.131} C_VEL
LIN {X 0,Y 178.8,Z 462.083,A -85,B 0,C 180,E1 -23162.552,E2 -23162.552} C_VEL
LIN {X 0,Y 180.29,Z 450.726,A -85,B 0,C 180,E1 -23163.563,E2 -23163.563} C_VEL
LIN {X 0,Y 181.36,Z 438.065,A -85,B 0,C 180,E1 -23164.305,E2 -23164.305} C_VEL
LIN {X 0,Y 183.475,Z 393.392,A -85,B 0,C 180,E1 -23165.966,E2 -23165.966} C_VEL
LIN {X 0,Y 181.201,Z 370.003,A -85,B 0,C 180,E1 -23167.448,E2 -23167.448} C_VEL
LIN {X 0,Y 174.188,Z 351.602,A -85,B 0,C 180,E1 -23169.746,E2 -23169.746} C_VEL
LIN {X 0,Y 168.465,Z 339.391,A -85,B 0,C 180,E1 -23171.668,E2 -23171.668} C_VEL
LIN {X 0,Y 164.713,Z 331.743,A -85,B 0,C 180,E1 -23173.059,E2 -23173.059} C_VEL
LIN {X 0,Y 164.285,Z 330.02,A -85,B 0,C 180,E1 -23174.229,E2 -23174.229} C_VEL
LIN {X 0,Y 164.271,Z 330.02,A -85,B 0,C 180,E1 -23176.801,E2 -23176.801} C_VEL
LIN {X 0,Y 164.303,Z 330.015,A -85,B 0,C 180,E1 -23180.354,E2 -23180.354} C_VEL
LIN {X 0,Y 164.339,Z 330.011,A -85,B 0,C 180,E1 -23184.35,E2 -23184.35} C_VEL
LIN {X 0,Y 164.4,Z 330,A -85,B 0,C 180,E1 -23189.136,E2 -23189.136} C_VEL
LIN {X 0,Y 164.415,Z 330.004,A -85,B 0,C 180,E1 -23194.693,E2 -23194.693} C_VEL
LIN {X 0,Y 164.426,Z 329.984,A -85,B 0,C 180,E1 -23200.117,E2 -23200.117} C_VEL
LIN {X 0,Y 164.495,Z 329.987,A -85,B 0,C 180,E1 -23205.146,E2 -23205.146} C_VEL
LIN {X 0,Y 164.773,Z 329.947,A -85,B 0,C 180,E1 -23210.176,E2 -23210.176} C_VEL
LIN {X 0,Y 164.831,Z 329.918,A -85,B 0,C 180,E1 -23212.65,E2 -23212.65} C_VEL
LIN {X 0,Y 165.051,Z 329.918,A -85,B 0,C 180,E1 -23217.559,E2 -23217.559} C_VEL
LIN {X 0,Y 165.301,Z 329.892,A -85,B 0,C 180,E1 -23219.999,E2 -23219.999} C_VEL
LIN {X 0,Y 164.766,Z 329.923,A -85,B 0,C 180,E1 -23224.893,E2 -23224.893} C_VEL
LIN {X 0,Y 164.837,Z 329.918,A -85,B 0,C 180,E1 -23227.348,E2 -23227.348} C_VEL
LIN {X 0,Y 164.711,Z 329.966,A -85,B 0,C 180,E1 -23231.059,E2 -23231.059} C_VEL
LIN {X 0,Y 164.46,Z 329.997,A -85,B 0,C 180,E1 -23237.405,E2 -23237.405} C_VEL
LIN {X 0,Y 164.457,Z 329.998,A -85,B 0,C 180,E1 -23239.991,E2 -23239.991} C_VEL
LIN {X 0,Y 164.394,Z 330.005,A -85,B 0,C 180,E1 -23246.126,E2 -23246.126} C_VEL
LIN {X 0,Y 164.383,Z 330.006,A -85,B 0,C 180,E1 -23251.226,E2 -23251.226} C_VEL
LIN {X 0,Y 164.301,Z 330.013,A -85,B 0,C 180,E1 -23256.787,E2 -23256.787} C_VEL
LIN {X 0,Y 164.297,Z 330.007,A -85,B 0,C 180,E1 -23259.914,E2 -23259.914} C_VEL
LIN {X 0,Y 164.285,Z 330.018,A -85,B 0,C 180,E1 -23263.339,E2 -23263.339} C_VEL
LIN {X 0,Y 164.269,Z 330.018,A -85,B 0,C 180,E1 -23266.796,E2 -23266.796} C_VEL
LIN {X 0,Y 164.3,Z 330.011,A -85,B 0,C 180,E1 -23270.349,E2 -23270.349} C_VEL
LIN {X 0,Y 164.335,Z 330.009,A -85,B 0,C 180,E1 -23274.346,E2 -23274.346} C_VEL
LIN {X 0,Y 164.393,Z 330.004,A -85,B 0,C 180,E1 -23279.131,E2 -23279.131} C_VEL
LIN {X 0,Y 164.366,Z 330.008,A -85,B 0,C 180,E1 -23282.398,E2 -23282.398} C_VEL
LIN {X 0,Y 165.311,Z 332.745,A -85,B 0,C 180,E1 -23282.812,E2 -23282.812} C_VEL
LIN {X 0,Y 167.038,Z 335.223,A -85,B 0,C 180,E1 -23283.374,E2 -23283.374} C_VEL
LIN {X 0,Y 173.035,Z 345.634,A -85,B 0,C 180,E1 -23285.311,E2 -23285.311} C_VEL
LIN {X 0,Y 179.597,Z 358.507,A -85,B 0,C 180,E1 -23287.312,E2 -23287.312} C_VEL
LIN {X 0,Y 183.718,Z 368.399,A -85,B 0,C 180,E1 -23288.558,E2 -23288.558} C_VEL
LIN {X 0,Y 184.434,Z 370.562,A -85,B 0,C 180,E1 -23288.787,E2 -23288.787} C_VEL
LIN {X 0,Y 181.4,Z 429.405,A -85,B 0,C 180,E1 -23290.959,E2 -23290.959} C_VEL
LIN {X 0,Y 180.088,Z 442.852,A -85,B 0,C 180,E1 -23291.878,E2 -23291.878} C_VEL
LIN {X 0,Y 178.455,Z 455.898,A -85,B 0,C 180,E1 -23293.259,E2 -23293.259} C_VEL
LIN {X 0,Y 176.193,Z 467.827,A -85,B 0,C 180,E1 -23294.97,E2 -23294.97} C_VEL
LIN {X 0,Y 173.945,Z 479.192,A -85,B 0,C 180,E1 -23297.157,E2 -23297.157} C_VEL
LIN {X 0,Y 171.476,Z 489.338,A -85,B 0,C 180,E1 -23299.621,E2 -23299.621} C_VEL
LIN {X 0,Y 169.252,Z 497.915,A -85,B 0,C 180,E1 -23302.241,E2 -23302.241} C_VEL
LIN {X 0,Y 166.719,Z 507.059,A -85,B 0,C 180,E1 -23305.766,E2 -23305.766} C_VEL
LIN {X 0,Y 164.8,Z 514.417,A -85,B 0,C 180,E1 -23309.385,E2 -23309.385} C_VEL
LIN {X 0,Y 163.627,Z 519.39,A -85,B 0,C 180,E1 -23312.458,E2 -23312.458} C_VEL
LIN {X 0,Y 162.633,Z 524.373,A -85,B 0,C 180,E1 -23316.325,E2 -23316.325} C_VEL
LIN {X 0,Y 161.879,Z 527.957,A -85,B 0,C 180,E1 -23319.997,E2 -23319.997} C_VEL
LIN {X 0,Y 161.613,Z 529.882,A -85,B 0,C 180,E1 -23322.554,E2 -23322.554} C_VEL
LIN {X 0,Y 161.69,Z 532.12,A -85,B 0,C 180,E1 -23327.012,E2 -23327.012} C_VEL
LIN {X 0,Y 162.07,Z 532.979,A -85,B 0,C 180,E1 -23330.294,E2 -23330.294} C_VEL
LIN {X 0,Y 162.625,Z 533.16,A -85,B 0,C 180,E1 -23332.884,E2 -23332.884} C_VEL
LIN {X 0,Y 163.461,Z 532.909,A -85,B 0,C 180,E1 -23335.46,E2 -23335.46} C_VEL
LIN {X 0,Y 164.514,Z 532.251,A -85,B 0,C 180,E1 -23338.024,E2 -23338.024} C_VEL
LIN {X 0,Y 165.85,Z 531.157,A -85,B 0,C 180,E1 -23340.56,E2 -23340.56} C_VEL
LIN {X 0,Y 168.389,Z 528.646,A -85,B 0,C 180,E1 -23344.29,E2 -23344.29} C_VEL
LIN {X 0,Y 171.582,Z 525.039,A -85,B 0,C 180,E1 -23347.903,E2 -23347.903} C_VEL
LIN {X 0,Y 175.384,Z 520.219,A -85,B 0,C 180,E1 -23351.385,E2 -23351.385} C_VEL
LIN {X 0,Y 179.763,Z 514.031,A -85,B 0,C 180,E1 -23354.721,E2 -23354.721} C_VEL
LIN {X 0,Y 184.67,Z 506.24,A -85,B 0,C 180,E1 -23357.906,E2 -23357.906} C_VEL
LIN {X 0,Y 189.197,Z 498.188,A -85,B 0,C 180,E1 -23360.419,E2 -23360.419} C_VEL
LIN {X 0,Y 194.094,Z 488.235,A -85,B 0,C 180,E1 -23362.801,E2 -23362.801} C_VEL
LIN {X 0,Y 198.608,Z 477.281,A -85,B 0,C 180,E1 -23364.838,E2 -23364.838} C_VEL
LIN {X 0,Y 202.448,Z 466.052,A -85,B 0,C 180,E1 -23366.418,E2 -23366.418} C_VEL
LIN {X 0,Y 205.719,Z 453.786,A -85,B 0,C 180,E1 -23367.723,E2 -23367.723} C_VEL
LIN {X 0,Y 208.357,Z 440.607,A -85,B 0,C 180,E1 -23368.712,E2 -23368.712} C_VEL
LIN {X 0,Y 210.022,Z 427.634,A -85,B 0,C 180,E1 -23369.324,E2 -23369.324} C_VEL
LIN {X 0,Y 212.297,Z 396.172,A -85,B 0,C 180,E1 -23370.296,E2 -23370.296} C_VEL
LIN {X 0,Y 207.964,Z 387.054,A -85,B 0,C 180,E1 -23372.38,E2 -23372.38} C_VEL
LIN {X 0,Y 202.642,Z 378.139,A -85,B 0,C 180,E1 -23375.08,E2 -23375.08} C_VEL
LIN {X 0,Y 197.301,Z 370.019,A -85,B 0,C 180,E1 -23378.106,E2 -23378.106} C_VEL
LIN {X 0,Y 194.488,Z 366.119,A -85,B 0,C 180,E1 -23379.857,E2 -23379.857} C_VEL
LIN {X 0,Y 191.74,Z 362.28,A -85,B 0,C 180,E1 -23381.755,E2 -23381.755} C_VEL
LIN {X 0,Y 188.426,Z 357.752,A -85,B 0,C 180,E1 -23384.312,E2 -23384.312} C_VEL
LIN {X 0,Y 185.719,Z 354.262,A -85,B 0,C 180,E1 -23386.668,E2 -23386.668} C_VEL
LIN {X 0,Y 184.974,Z 353.141,A -85,B 0,C 180,E1 -23387.393,E2 -23387.393} C_VEL
LIN {X 0,Y 182.354,Z 350.441,A -85,B 0,C 180,E1 -23390.06,E2 -23390.06} C_VEL
LIN {X 0,Y 180.936,Z 347.762,A -85,B 0,C 180,E1 -23391.906,E2 -23391.906} C_VEL
LIN {X 0,Y 178.032,Z 345.496,A -85,B 0,C 180,E1 -23396.11,E2 -23396.11} C_VEL
LIN {X 0,Y 176.928,Z 342.86,A -85,B 0,C 180,E1 -23398.72,E2 -23398.72} C_VEL
LIN {X 0,Y 176.703,Z 342.072,A -85,B 0,C 180,E1 -23399.431,E2 -23399.431} C_VEL
LIN {X 0,Y 175.145,Z 341.713,A -85,B 0,C 180,E1 -23409.237,E2 -23409.237} C_VEL
LIN {X 0,Y 176.475,Z 342.343,A -85,B 0,C 180,E1 -23414.652,E2 -23414.652} C_VEL
LIN {X 0,Y 177.491,Z 345.012,A -85,B 0,C 180,E1 -23417.425,E2 -23417.425} C_VEL
LIN {X 0,Y 179.688,Z 347.374,A -85,B 0,C 180,E1 -23421.096,E2 -23421.096} C_VEL
LIN {X 0,Y 180.8,Z 348.238,A -85,B 0,C 180,E1 -23422.547,E2 -23422.547} C_VEL
LIN {X 0,Y 186.142,Z 355.871,A -85,B 0,C 180,E1 -23428.373,E2 -23428.373} C_VEL
LIN {X 0,Y 190.357,Z 362.334,A -85,B 0,C 180,E1 -23431.933,E2 -23431.933} C_VEL
LIN {X 0,Y 193.847,Z 368.096,A -85,B 0,C 180,E1 -23434.482,E2 -23434.482} C_VEL
LIN {X 0,Y 196.871,Z 373.264,A -85,B 0,C 180,E1 -23436.451,E2 -23436.451} C_VEL
LIN {X 0,Y 201.27,Z 381.126,A -85,B 0,C 180,E1 -23439.053,E2 -23439.053} C_VEL
LIN {X 0,Y 205.559,Z 389.953,A -85,B 0,C 180,E1 -23441.398,E2 -23441.398} C_VEL
LIN {X 0,Y 209.609,Z 399.357,A -85,B 0,C 180,E1 -23443.473,E2 -23443.473} C_VEL
LIN {X 0,Y 211.689,Z 404.677,A -85,B 0,C 180,E1 -23444.499,E2 -23444.499} C_VEL
LIN {X 0,Y 209.111,Z 440.256,A -85,B 0,C 180,E1 -23445.634,E2 -23445.634} C_VEL
LIN {X 0,Y 207.044,Z 453.783,A -85,B 0,C 180,E1 -23446.321,E2 -23446.321} C_VEL
LIN {X 0,Y 204.118,Z 466.83,A -85,B 0,C 180,E1 -23447.328,E2 -23447.328} C_VEL
LIN {X 0,Y 200.466,Z 478.625,A -85,B 0,C 180,E1 -23448.573,E2 -23448.573} C_VEL
LIN {X 0,Y 196.23,Z 489.968,A -85,B 0,C 180,E1 -23450.198,E2 -23450.198} C_VEL
LIN {X 0,Y 191.67,Z 500.228,A -85,B 0,C 180,E1 -23452.113,E2 -23452.113} C_VEL
LIN {X 0,Y 186.925,Z 509.472,A -85,B 0,C 180,E1 -23454.359,E2 -23454.359} C_VEL
LIN {X 0,Y 181.748,Z 518.455,A -85,B 0,C 180,E1 -23457.228,E2 -23457.228} C_VEL
LIN {X 0,Y 178.217,Z 523.91,A -85,B 0,C 180,E1 -23459.409,E2 -23459.409} C_VEL
LIN {X 0,Y 175.473,Z 527.067,A -85,B 0,C 180,E1 -23460.787,E2 -23460.787} C_VEL
LIN {X 0,Y 169.667,Z 531.736,A -85,B 0,C 180,E1 -23462.977,E2 -23462.977} C_VEL
LIN {X 0,Y 164.132,Z 535.677,A -85,B 0,C 180,E1 -23465.44,E2 -23465.44} C_VEL
LIN {X 0,Y 161.875,Z 537.682,A -85,B 0,C 180,E1 -23467.217,E2 -23467.217} C_VEL
LIN {X 0,Y 160.085,Z 539.738,A -85,B 0,C 180,E1 -23469.443,E2 -23469.443} C_VEL
LIN {X 0,Y 158.377,Z 541.512,A -85,B 0,C 180,E1 -23471.907,E2 -23471.907} C_VEL
LIN {X 0,Y 156.126,Z 543.867,A -85,B 0,C 180,E1 -23476.997,E2 -23476.997} C_VEL
LIN {X 0,Y 155.43,Z 544.477,A -85,B 0,C 180,E1 -23479.584,E2 -23479.584} C_VEL
LIN {X 0,Y 154.84,Z 544.476,A -85,B 0,C 180,E1 -23484.796,E2 -23484.796} C_VEL
LIN {X 0,Y 154.845,Z 543.894,A -85,B 0,C 180,E1 -23487.403,E2 -23487.403} C_VEL
LIN {X 0,Y 154.987,Z 542.922,A -85,B 0,C 180,E1 -23490.004,E2 -23490.004} C_VEL
LIN {X 0,Y 154.834,Z 541.21,A -85,B 0,C 180,E1 -23493.03,E2 -23493.03} C_VEL
LIN {X 0,Y 155.038,Z 537.277,A -85,B 0,C 180,E1 -23497.82,E2 -23497.82} C_VEL
LIN {X 0,Y 155.624,Z 532.835,A -85,B 0,C 180,E1 -23501.729,E2 -23501.729} C_VEL
LIN {X 0,Y 156.751,Z 527.159,A -85,B 0,C 180,E1 -23505.609,E2 -23505.609} C_VEL
LIN {X 0,Y 158.644,Z 520.048,A -85,B 0,C 180,E1 -23509.409,E2 -23509.409} C_VEL
LIN {X 0,Y 160.637,Z 512.768,A -85,B 0,C 180,E1 -23512.512,E2 -23512.512} C_VEL
LIN {X 0,Y 161.915,Z 507.847,A -85,B 0,C 180,E1 -23514.283,E2 -23514.283} C_VEL
LIN {X 0,Y 164.388,Z 498.765,A -85,B 0,C 180,E1 -23517.02,E2 -23517.02} C_VEL
LIN {X 0,Y 166.741,Z 489.161,A -85,B 0,C 180,E1 -23519.343,E2 -23519.343} C_VEL
LIN {X 0,Y 169.203,Z 478.896,A -85,B 0,C 180,E1 -23521.282,E2 -23521.282} C_VEL
LIN {X 0,Y 171.615,Z 466.728,A -85,B 0,C 180,E1 -23523.04,E2 -23523.04} C_VEL
LIN {X 0,Y 173.538,Z 453.909,A -85,B 0,C 180,E1 -23524.368,E2 -23524.368} C_VEL
LIN {X 0,Y 174.943,Z 441.1,A -85,B 0,C 180,E1 -23525.239,E2 -23525.239} C_VEL
LIN {X 0,Y 177.284,Z 393.836,A -85,B 0,C 180,E1 -23527.087,E2 -23527.087} C_VEL
LIN {X 0,Y 175.306,Z 372.374,A -85,B 0,C 180,E1 -23528.5,E2 -23528.5} C_VEL
LIN {X 0,Y 168.801,Z 355.073,A -85,B 0,C 180,E1 -23530.778,E2 -23530.778} C_VEL
LIN {X 0,Y 162.053,Z 340.498,A -85,B 0,C 180,E1 -23533.212,E2 -23533.212} C_VEL
LIN {X 0,Y 157.515,Z 332.1,A -85,B 0,C 180,E1 -23534.928,E2 -23534.928} C_VEL
LIN {X 0,Y 157.311,Z 331.329,A -85,B 0,C 180,E1 -23535.141,E2 -23535.141} C_VEL
LIN {X 0,Y 157.224,Z 330.9,A -85,B 0,C 180,E1 -23535.665,E2 -23535.665} C_VEL
LIN {X 0,Y 157.214,Z 330.898,A -85,B 0,C 180,E1 -23541.255,E2 -23541.255} C_VEL
LIN {X 0,Y 157.287,Z 330.89,A -85,B 0,C 180,E1 -23544.487,E2 -23544.487} C_VEL
LIN {X 0,Y 157.302,Z 330.888,A -85,B 0,C 180,E1 -23548.097,E2 -23548.097} C_VEL
LIN {X 0,Y 157.324,Z 330.887,A -85,B 0,C 180,E1 -23553.466,E2 -23553.466} C_VEL
LIN {X 0,Y 157.37,Z 330.866,A -85,B 0,C 180,E1 -23559.701,E2 -23559.701} C_VEL
LIN {X 0,Y 157.427,Z 330.861,A -85,B 0,C 180,E1 -23564.463,E2 -23564.463} C_VEL
LIN {X 0,Y 157.695,Z 330.831,A -85,B 0,C 180,E1 -23569.731,E2 -23569.731} C_VEL
LIN {X 0,Y 157.769,Z 330.798,A -85,B 0,C 180,E1 -23572.32,E2 -23572.32} C_VEL
LIN {X 0,Y 158.264,Z 330.769,A -85,B 0,C 180,E1 -23579.999,E2 -23579.999} C_VEL
LIN {X 0,Y 157.774,Z 330.8,A -85,B 0,C 180,E1 -23587.679,E2 -23587.679} C_VEL
LIN {X 0,Y 157.641,Z 330.846,A -85,B 0,C 180,E1 -23591.227,E2 -23591.227} C_VEL
LIN {X 0,Y 157.43,Z 330.863,A -85,B 0,C 180,E1 -23595.536,E2 -23595.536} C_VEL
LIN {X 0,Y 157.365,Z 330.877,A -85,B 0,C 180,E1 -23600.933,E2 -23600.933} C_VEL
LIN {X 0,Y 157.317,Z 330.886,A -85,B 0,C 180,E1 -23606.679,E2 -23606.679} C_VEL
LIN {X 0,Y 157.283,Z 330.889,A -85,B 0,C 180,E1 -23612.425,E2 -23612.425} C_VEL
LIN {X 0,Y 157.275,Z 330.887,A -85,B 0,C 180,E1 -23616.447,E2 -23616.447} C_VEL
LIN {X 0,Y 157.199,Z 330.899,A -85,B 0,C 180,E1 -23622.114,E2 -23622.114} C_VEL
LIN {X 0,Y 157.198,Z 330.903,A -85,B 0,C 180,E1 -23627.881,E2 -23627.881} C_VEL
LIN {X 0,Y 157.273,Z 330.892,A -85,B 0,C 180,E1 -23633.548,E2 -23633.548} C_VEL
LIN {X 0,Y 157.35,Z 330.882,A -85,B 0,C 180,E1 -23639.345,E2 -23639.345} C_VEL
LIN {X 0,Y 157.305,Z 331.1,A -85,B 0,C 180,E1 -23640.56,E2 -23640.56} C_VEL
LIN {X 0,Y 158.407,Z 333.939,A -85,B 0,C 180,E1 -23641.038,E2 -23641.038} C_VEL
LIN {X 0,Y 159.985,Z 336.042,A -85,B 0,C 180,E1 -23641.594,E2 -23641.594} C_VEL
LIN {X 0,Y 166.96,Z 347.798,A -85,B 0,C 180,E1 -23644.016,E2 -23644.016} C_VEL
LIN {X 0,Y 174.036,Z 361.717,A -85,B 0,C 180,E1 -23646.323,E2 -23646.323} C_VEL
LIN {X 0,Y 178.124,Z 371.621,A -85,B 0,C 180,E1 -23647.638,E2 -23647.638} C_VEL
LIN {X 0,Y 177.79,Z 381.934,A -85,B 0,C 180,E1 -23648.058,E2 -23648.058} C_VEL
LIN {X 0,Y 175.163,Z 429.777,A -85,B 0,C 180,E1 -23649.878,E2 -23649.878} C_VEL
LIN {X 0,Y 173.812,Z 442.998,A -85,B 0,C 180,E1 -23650.804,E2 -23650.804} C_VEL
LIN {X 0,Y 172.166,Z 455.632,A -85,B 0,C 180,E1 -23652.169,E2 -23652.169} C_VEL
LIN {X 0,Y 169.994,Z 466.898,A -85,B 0,C 180,E1 -23653.792,E2 -23653.792} C_VEL
LIN {X 0,Y 167.578,Z 478.492,A -85,B 0,C 180,E1 -23656.042,E2 -23656.042} C_VEL
LIN {X 0,Y 165.128,Z 488.314,A -85,B 0,C 180,E1 -23658.454,E2 -23658.454} C_VEL
LIN {X 0,Y 162.647,Z 497.535,A -85,B 0,C 180,E1 -23661.298,E2 -23661.298} C_VEL
LIN {X 0,Y 160.388,Z 505.433,A -85,B 0,C 180,E1 -23664.338,E2 -23664.338} C_VEL
LIN {X 0,Y 158.207,Z 513.134,A -85,B 0,C 180,E1 -23668.087,E2 -23668.087} C_VEL
LIN {X 0,Y 156.898,Z 518.395,A -85,B 0,C 180,E1 -23671.28,E2 -23671.28} C_VEL
LIN {X 0,Y 155.773,Z 523.493,A -85,B 0,C 180,E1 -23675.173,E2 -23675.173} C_VEL
LIN {X 0,Y 154.92,Z 527.467,A -85,B 0,C 180,E1 -23679.132,E2 -23679.132} C_VEL
LIN {X 0,Y 154.493,Z 530.391,A -85,B 0,C 180,E1 -23683.143,E2 -23683.143} C_VEL
LIN {X 0,Y 154.626,Z 532.378,A -85,B 0,C 180,E1 -23687.354,E2 -23687.354} C_VEL
LIN {X 0,Y 155.144,Z 533.305,A -85,B 0,C 180,E1 -23691.243,E2 -23691.243} C_VEL
LIN {X 0,Y 156.578,Z 533.189,A -85,B 0,C 180,E1 -23696.144,E2 -23696.144} C_VEL
LIN {X 0,Y 157.944,Z 532.391,A -85,B 0,C 180,E1 -23699.301,E2 -23699.301} C_VEL
LIN {X 0,Y 160.762,Z 530.035,A -85,B 0,C 180,E1 -23703.838,E2 -23703.838} C_VEL
LIN {X 0,Y 164.502,Z 526.215,A -85,B 0,C 180,E1 -23708.273,E2 -23708.273} C_VEL
LIN {X 0,Y 168.412,Z 521.699,A -85,B 0,C 180,E1 -23711.884,E2 -23711.884} C_VEL
LIN {X 0,Y 172.883,Z 515.869,A -85,B 0,C 180,E1 -23715.344,E2 -23715.344} C_VEL
LIN {X 0,Y 177.967,Z 508.443,A -85,B 0,C 180,E1 -23718.612,E2 -23718.612} C_VEL
LIN {X 0,Y 182.567,Z 500.806,A -85,B 0,C 180,E1 -23721.212,E2 -23721.212} C_VEL
LIN {X 0,Y 187.979,Z 490.778,A -85,B 0,C 180,E1 -23723.807,E2 -23723.807} C_VEL
LIN {X 0,Y 192.326,Z 481.076,A -85,B 0,C 180,E1 -23725.761,E2 -23725.761} C_VEL
LIN {X 0,Y 196.808,Z 469.218,A -85,B 0,C 180,E1 -23727.563,E2 -23727.563} C_VEL
LIN {X 0,Y 200.383,Z 457.055,A -85,B 0,C 180,E1 -23728.985,E2 -23728.985} C_VEL
LIN {X 0,Y 203.244,Z 444.409,A -85,B 0,C 180,E1 -23730.005,E2 -23730.005} C_VEL
LIN {X 0,Y 205.256,Z 431.304,A -85,B 0,C 180,E1 -23730.717,E2 -23730.717} C_VEL
LIN {X 0,Y 207.812,Z 399.012,A -85,B 0,C 180,E1 -23731.741,E2 -23731.741} C_VEL
LIN {X 0,Y 204.347,Z 391.727,A -85,B 0,C 180,E1 -23733.514,E2 -23733.514} C_VEL
LIN {X 0,Y 199.798,Z 383.87,A -85,B 0,C 180,E1 -23735.959,E2 -23735.959} C_VEL
LIN {X 0,Y 194.526,Z 375.646,A -85,B 0,C 180,E1 -23739.111,E2 -23739.111} C_VEL
LIN {X 0,Y 192.298,Z 372.405,A -85,B 0,C 180,E1 -23740.589,E2 -23740.589} C_VEL
LIN {X 0,Y 189.679,Z 368.621,A -85,B 0,C 180,E1 -23742.493,E2 -23742.493} C_VEL
LIN {X 0,Y 186.437,Z 364.088,A -85,B 0,C 180,E1 -23745.12,E2 -23745.12} C_VEL
LIN {X 0,Y 183.707,Z 360.277,A -85,B 0,C 180,E1 -23747.662,E2 -23747.662} C_VEL
LIN {X 0,Y 180.468,Z 356.453,A -85,B 0,C 180,E1 -23751.18,E2 -23751.18} C_VEL
LIN {X 0,Y 179.599,Z 354.639,A -85,B 0,C 180,E1 -23752.411,E2 -23752.411} C_VEL
LIN {X 0,Y 176.806,Z 352.232,A -85,B 0,C 180,E1 -23756.725,E2 -23756.725} C_VEL
LIN {X 0,Y 175.748,Z 349.437,A -85,B 0,C 180,E1 -23759.5,E2 -23759.5} C_VEL
LIN {X 0,Y 175.59,Z 349.04,A -85,B 0,C 180,E1 -23760,E2 -23760} C_VEL
LIN {X 0,Y 174.27,Z 348.762,A -85,B 0,C 180,E1 -23769.284,E2 -23769.284} C_VEL
LIN {X 0,Y 175.426,Z 349.41,A -85,B 0,C 180,E1 -23774.242,E2 -23774.242} C_VEL
LIN {X 0,Y 177.026,Z 352.9,A -85,B 0,C 180,E1 -23778.327,E2 -23778.327} C_VEL
LIN {X 0,Y 179.568,Z 355.121,A -85,B 0,C 180,E1 -23782.161,E2 -23782.161} C_VEL
LIN {X 0,Y 184.335,Z 362.351,A -85,B 0,C 180,E1 -23787.626,E2 -23787.626} C_VEL
LIN {X 0,Y 188.138,Z 368.369,A -85,B 0,C 180,E1 -23791.021,E2 -23791.021} C_VEL
LIN {X 0,Y 191.642,Z 374.409,A -85,B 0,C 180,E1 -23793.736,E2 -23793.736} C_VEL
LIN {X 0,Y 194.941,Z 380.359,A -85,B 0,C 180,E1 -23795.991,E2 -23795.991} C_VEL
LIN {X 0,Y 198.792,Z 387.635,A -85,B 0,C 180,E1 -23798.373,E2 -23798.373} C_VEL
LIN {X 0,Y 203.268,Z 397.377,A -85,B 0,C 180,E1 -23800.934,E2 -23800.934} C_VEL
LIN {X 0,Y 207.253,Z 407.419,A -85,B 0,C 180,E1 -23803.075,E2 -23803.075} C_VEL
LIN {X 0,Y 204.585,Z 440.899,A -85,B 0,C 180,E1 -23804.131,E2 -23804.131} C_VEL
LIN {X 0,Y 202.371,Z 454.472,A -85,B 0,C 180,E1 -23804.835,E2 -23804.835} C_VEL
LIN {X 0,Y 199.295,Z 467.37,A -85,B 0,C 180,E1 -23805.861,E2 -23805.861} C_VEL
LIN {X 0,Y 195.236,Z 479.77,A -85,B 0,C 180,E1 -23807.204,E2 -23807.204} C_VEL
LIN {X 0,Y 190.853,Z 490.847,A -85,B 0,C 180,E1 -23808.84,E2 -23808.84} C_VEL
LIN {X 0,Y 186.153,Z 500.849,A -85,B 0,C 180,E1 -23810.779,E2 -23810.779} C_VEL
LIN {X 0,Y 181.227,Z 509.912,A -85,B 0,C 180,E1 -23813.057,E2 -23813.057} C_VEL
LIN {X 0,Y 175.836,Z 518.773,A -85,B 0,C 180,E1 -23815.979,E2 -23815.979} C_VEL
LIN {X 0,Y 170.862,Z 525.939,A -85,B 0,C 180,E1 -23819.063,E2 -23819.063} C_VEL
LIN {X 0,Y 166.702,Z 531.684,A -85,B 0,C 180,E1 -23822.375,E2 -23822.375} C_VEL
LIN {X 0,Y 163.133,Z 536.242,A -85,B 0,C 180,E1 -23825.845,E2 -23825.845} C_VEL
LIN {X 0,Y 161.875,Z 537.682,A -85,B 0,C 180,E1 -23827.217,E2 -23827.217} C_VEL
LIN {X 0,Y 159.721,Z 539.483,A -85,B 0,C 180,E1 -23829.076,E2 -23829.076} C_VEL
LIN {X 0,Y 154.768,Z 541.796,A -85,B 0,C 180,E1 -23832.091,E2 -23832.091} C_VEL
LIN {X 0,Y 150.238,Z 543.372,A -85,B 0,C 180,E1 -23835.35,E2 -23835.35} C_VEL
LIN {X 0,Y 148.809,Z 543.927,A -85,B 0,C 180,E1 -23837.531,E2 -23837.531} C_VEL
LIN {X 0,Y 147.937,Z 544.392,A -85,B 0,C 180,E1 -23841.811,E2 -23841.811} C_VEL
LIN {X 0,Y 147.748,Z 544.158,A -85,B 0,C 180,E1 -23844.545,E2 -23844.545} C_VEL
LIN {X 0,Y 147.756,Z 543.542,A -85,B 0,C 180,E1 -23847.278,E2 -23847.278} C_VEL
LIN {X 0,Y 147.894,Z 542.533,A -85,B 0,C 180,E1 -23850.004,E2 -23850.004} C_VEL
LIN {X 0,Y 147.757,Z 541.042,A -85,B 0,C 180,E1 -23852.73,E2 -23852.73} C_VEL
LIN {X 0,Y 147.862,Z 537.995,A -85,B 0,C 180,E1 -23856.828,E2 -23856.828} C_VEL
LIN {X 0,Y 148.371,Z 533.854,A -85,B 0,C 180,E1 -23860.926,E2 -23860.926} C_VEL
LIN {X 0,Y 149.604,Z 527.474,A -85,B 0,C 180,E1 -23865.675,E2 -23865.675} C_VEL
LIN {X 0,Y 151.556,Z 520.528,A -85,B 0,C 180,E1 -23869.649,E2 -23869.649} C_VEL
LIN {X 0,Y 153.622,Z 513.408,A -85,B 0,C 180,E1 -23872.888,E2 -23872.888} C_VEL
LIN {X 0,Y 155.105,Z 507.842,A -85,B 0,C 180,E1 -23875.01,E2 -23875.01} C_VEL
LIN {X 0,Y 157.743,Z 498.647,A -85,B 0,C 180,E1 -23877.896,E2 -23877.896} C_VEL
LIN {X 0,Y 160.188,Z 489.07,A -85,B 0,C 180,E1 -23880.305,E2 -23880.305} C_VEL
LIN {X 0,Y 163.184,Z 477.239,A -85,B 0,C 180,E1 -23882.575,E2 -23882.575} C_VEL
LIN {X 0,Y 165.492,Z 465.64,A -85,B 0,C 180,E1 -23884.246,E2 -23884.246} C_VEL
LIN {X 0,Y 167.497,Z 452.534,A -85,B 0,C 180,E1 -23885.608,E2 -23885.608} C_VEL
LIN {X 0,Y 168.86,Z 439.881,A -85,B 0,C 180,E1 -23886.463,E2 -23886.463} C_VEL
LIN {X 0,Y 171.185,Z 394.691,A -85,B 0,C 180,E1 -23888.263,E2 -23888.263} C_VEL
LIN {X 0,Y 169.432,Z 374.749,A -85,B 0,C 180,E1 -23889.633,E2 -23889.633} C_VEL
LIN {X 0,Y 163.624,Z 358.9,A -85,B 0,C 180,E1 -23891.815,E2 -23891.815} C_VEL
LIN {X 0,Y 157.621,Z 345.681,A -85,B 0,C 180,E1 -23894.118,E2 -23894.118} C_VEL
LIN {X 0,Y 153.48,Z 337.936,A -85,B 0,C 180,E1 -23895.775,E2 -23895.775} C_VEL
LIN {X 0,Y 152.236,Z 335.964,A -85,B 0,C 180,E1 -23896.276,E2 -23896.276} C_VEL
LIN {X 0,Y 150.612,Z 333.541,A -85,B 0,C 180,E1 -23896.939,E2 -23896.939} C_VEL
LIN {X 0,Y 150.14,Z 331.781,A -85,B 0,C 180,E1 -23897.29,E2 -23897.29} C_VEL
LIN {X 0,Y 150.187,Z 331.77,A -85,B 0,C 180,E1 -23902.709,E2 -23902.709} C_VEL
LIN {X 0,Y 150.224,Z 331.768,A -85,B 0,C 180,E1 -23907.369,E2 -23907.369} C_VEL
LIN {X 0,Y 150.25,Z 331.769,A -85,B 0,C 180,E1 -23912.722,E2 -23912.722} C_VEL
LIN {X 0,Y 150.294,Z 331.75,A -85,B 0,C 180,E1 -23919.275,E2 -23919.275} C_VEL
LIN {X 0,Y 150.331,Z 331.737,A -85,B 0,C 180,E1 -23923.709,E2 -23923.709} C_VEL
LIN {X 0,Y 150.616,Z 331.716,A -85,B 0,C 180,E1 -23929.242,E2 -23929.242} C_VEL
LIN {X 0,Y 150.691,Z 331.68,A -85,B 0,C 180,E1 -23931.956,E2 -23931.956} C_VEL
LIN {X 0,Y 151.224,Z 331.645,A -85,B 0,C 180,E1 -23939.999,E2 -23939.999} C_VEL
LIN {X 0,Y 150.712,Z 331.681,A -85,B 0,C 180,E1 -23948.041,E2 -23948.041} C_VEL
LIN {X 0,Y 150.583,Z 331.725,A -85,B 0,C 180,E1 -23951.43,E2 -23951.43} C_VEL
LIN {X 0,Y 150.337,Z 331.747,A -85,B 0,C 180,E1 -23956.289,E2 -23956.289} C_VEL
LIN {X 0,Y 150.347,Z 331.752,A -85,B 0,C 180,E1 -23960.778,E2 -23960.778} C_VEL
LIN {X 0,Y 150.249,Z 331.763,A -85,B 0,C 180,E1 -23967.277,E2 -23967.277} C_VEL
LIN {X 0,Y 150.222,Z 331.769,A -85,B 0,C 180,E1 -23972.63,E2 -23972.63} C_VEL
LIN {X 0,Y 150.184,Z 331.774,A -85,B 0,C 180,E1 -23977.469,E2 -23977.469} C_VEL
LIN {X 0,Y 150.142,Z 331.772,A -85,B 0,C 180,E1 -23981.496,E2 -23981.496} C_VEL
LIN {X 0,Y 150.131,Z 331.774,A -85,B 0,C 180,E1 -23985.392,E2 -23985.392} C_VEL
LIN {X 0,Y 150.146,Z 331.778,A -85,B 0,C 180,E1 -23989.052,E2 -23989.052} C_VEL
LIN {X 0,Y 150.184,Z 331.777,A -85,B 0,C 180,E1 -23992.705,E2 -23992.705} C_VEL
LIN {X 0,Y 150.264,Z 331.763,A -85,B 0,C 180,E1 -23998.399,E2 -23998.399} C_VEL
LIN {X 0,Y 151.292,Z 334.618,A -85,B 0,C 180,E1 -23998.962,E2 -23998.962} C_VEL
LIN {X 0,Y 152.897,Z 336.719,A -85,B 0,C 180,E1 -23999.59,E2 -23999.59} C_VEL
LIN {X 0,Y 155.066,Z 340.192,A -85,B 0,C 180,E1 -24000.447,E2 -24000.447} C_VEL
LIN {X 0,Y 162.178,Z 352.307,A -85,B 0,C 180,E1 -24003.076,E2 -24003.076} C_VEL
LIN {X 0,Y 169.143,Z 366.333,A -85,B 0,C 180,E1 -24005.481,E2 -24005.481} C_VEL
LIN {X 0,Y 172.183,Z 373.874,A -85,B 0,C 180,E1 -24006.526,E2 -24006.526} C_VEL
LIN {X 0,Y 168.956,Z 430.457,A -85,B 0,C 180,E1 -24008.734,E2 -24008.734} C_VEL
LIN {X 0,Y 167.541,Z 443.683,A -85,B 0,C 180,E1 -24009.7,E2 -24009.7} C_VEL
LIN {X 0,Y 165.782,Z 456.432,A -85,B 0,C 180,E1 -24011.137,E2 -24011.137} C_VEL
LIN {X 0,Y 163.207,Z 469.136,A -85,B 0,C 180,E1 -24013.098,E2 -24013.098} C_VEL
LIN {X 0,Y 160.712,Z 480.369,A -85,B 0,C 180,E1 -24015.433,E2 -24015.433} C_VEL
LIN {X 0,Y 157.779,Z 491.265,A -85,B 0,C 180,E1 -24018.354,E2 -24018.354} C_VEL
LIN {X 0,Y 155.115,Z 500.499,A -85,B 0,C 180,E1 -24021.528,E2 -24021.528} C_VEL
LIN {X 0,Y 152.504,Z 509.28,A -85,B 0,C 180,E1 -24025.37,E2 -24025.37} C_VEL
LIN {X 0,Y 150.489,Z 516.275,A -85,B 0,C 180,E1 -24029.327,E2 -24029.327} C_VEL
LIN {X 0,Y 148.948,Z 522.69,A -85,B 0,C 180,E1 -24034.054,E2 -24034.054} C_VEL
LIN {X 0,Y 147.994,Z 526.92,A -85,B 0,C 180,E1 -24038.186,E2 -24038.186} C_VEL
LIN {X 0,Y 147.558,Z 529.15,A -85,B 0,C 180,E1 -24040.979,E2 -24040.979} C_VEL
LIN {X 0,Y 147.4,Z 530.895,A -85,B 0,C 180,E1 -24043.788,E2 -24043.788} C_VEL
LIN {X 0,Y 147.552,Z 532.63,A -85,B 0,C 180,E1 -24047.711,E2 -24047.711} C_VEL
LIN {X 0,Y 148.242,Z 533.607,A -85,B 0,C 180,E1 -24052.284,E2 -24052.284} C_VEL
LIN {X 0,Y 149.694,Z 533.473,A -85,B 0,C 180,E1 -24056.872,E2 -24056.872} C_VEL
LIN {X 0,Y 151.468,Z 532.492,A -85,B 0,C 180,E1 -24060.685,E2 -24060.685} C_VEL
LIN {X 0,Y 154.219,Z 530.357,A -85,B 0,C 180,E1 -24064.887,E2 -24064.887} C_VEL
LIN {X 0,Y 157.429,Z 527.36,A -85,B 0,C 180,E1 -24068.676,E2 -24068.676} C_VEL
LIN {X 0,Y 161.689,Z 522.838,A -85,B 0,C 180,E1 -24072.633,E2 -24072.633} C_VEL
LIN {X 0,Y 166.874,Z 516.547,A -85,B 0,C 180,E1 -24076.587,E2 -24076.587} C_VEL
LIN {X 0,Y 172.109,Z 509.385,A -85,B 0,C 180,E1 -24079.88,E2 -24079.88} C_VEL
LIN {X 0,Y 176.978,Z 501.739,A -85,B 0,C 180,E1 -24082.575,E2 -24082.575} C_VEL
LIN {X 0,Y 182.222,Z 492.555,A -85,B 0,C 180,E1 -24085.036,E2 -24085.036} C_VEL
LIN {X 0,Y 187.129,Z 482.356,A -85,B 0,C 180,E1 -24087.169,E2 -24087.169} C_VEL
LIN {X 0,Y 191.172,Z 472.359,A -85,B 0,C 180,E1 -24088.785,E2 -24088.785} C_VEL
LIN {X 0,Y 195.185,Z 460.019,A -85,B 0,C 180,E1 -24090.296,E2 -24090.296} C_VEL
LIN {X 0,Y 198.184,Z 448.135,A -85,B 0,C 180,E1 -24091.357,E2 -24091.357} C_VEL
LIN {X 0,Y 200.499,Z 435.179,A -85,B 0,C 180,E1 -24092.16,E2 -24092.16} C_VEL
LIN {X 0,Y 202.094,Z 419.519,A -85,B 0,C 180,E1 -24092.716,E2 -24092.716} C_VEL
LIN {X 0,Y 203.465,Z 401.89,A -85,B 0,C 180,E1 -24093.246,E2 -24093.246} C_VEL
LIN {X 0,Y 200.125,Z 395.014,A -85,B 0,C 180,E1 -24095.076,E2 -24095.076} C_VEL
LIN {X 0,Y 194.803,Z 385.898,A -85,B 0,C 180,E1 -24098.206,E2 -24098.206} C_VEL
LIN {X 0,Y 190.097,Z 378.632,A -85,B 0,C 180,E1 -24101.372,E2 -24101.372} C_VEL
LIN {X 0,Y 187.223,Z 374.432,A -85,B 0,C 180,E1 -24103.579,E2 -24103.579} C_VEL
LIN {X 0,Y 184.633,Z 370.585,A -85,B 0,C 180,E1 -24105.816,E2 -24105.816} C_VEL
LIN {X 0,Y 181.571,Z 366.294,A -85,B 0,C 180,E1 -24108.841,E2 -24108.841} C_VEL
LIN {X 0,Y 178.978,Z 363.049,A -85,B 0,C 180,E1 -24111.87,E2 -24111.87} C_VEL
LIN {X 0,Y 178.067,Z 361.386,A -85,B 0,C 180,E1 -24113.2,E2 -24113.2} C_VEL
LIN {X 0,Y 175.444,Z 358.692,A -85,B 0,C 180,E1 -24117.705,E2 -24117.705} C_VEL
LIN {X 0,Y 174.604,Z 356.037,A -85,B 0,C 180,E1 -24120.275,E2 -24120.275} C_VEL
LIN {X 0,Y 173.533,Z 355.898,A -85,B 0,C 180,E1 -24130.367,E2 -24130.367} C_VEL
LIN {X 0,Y 174.404,Z 356.378,A -85,B 0,C 180,E1 -24133.844,E2 -24133.844} C_VEL
LIN {X 0,Y 175.946,Z 359.855,A -85,B 0,C 180,E1 -24137.999,E2 -24137.999} C_VEL
LIN {X 0,Y 178.254,Z 361.949,A -85,B 0,C 180,E1 -24141.653,E2 -24141.653} C_VEL
LIN {X 0,Y 182.619,Z 368.903,A -85,B 0,C 180,E1 -24146.924,E2 -24146.924} C_VEL
LIN {X 0,Y 185.975,Z 374.459,A -85,B 0,C 180,E1 -24150.098,E2 -24150.098} C_VEL
LIN {X 0,Y 189.42,Z 380.673,A -85,B 0,C 180,E1 -24152.93,E2 -24152.93} C_VEL
LIN {X 0,Y 192.4,Z 386.308,A -85,B 0,C 180,E1 -24155.103,E2 -24155.103} C_VEL
LIN {X 0,Y 196.311,Z 394.092,A -85,B 0,C 180,E1 -24157.656,E2 -24157.656} C_VEL
LIN {X 0,Y 200.928,Z 404.814,A -85,B 0,C 180,E1 -24160.433,E2 -24160.433} C_VEL
LIN {X 0,Y 202.859,Z 409.99,A -85,B 0,C 180,E1 -24161.544,E2 -24161.544} C_VEL
LIN {X 0,Y 200.279,Z 440.962,A -85,B 0,C 180,E1 -24162.536,E2 -24162.536} C_VEL
LIN {X 0,Y 198.013,Z 454.361,A -85,B 0,C 180,E1 -24163.235,E2 -24163.235} C_VEL
LIN {X 0,Y 194.921,Z 466.924,A -85,B 0,C 180,E1 -24164.23,E2 -24164.23} C_VEL
LIN {X 0,Y 190.7,Z 479.366,A -85,B 0,C 180,E1 -24165.561,E2 -24165.561} C_VEL
LIN {X 0,Y 186.168,Z 490.467,A -85,B 0,C 180,E1 -24167.199,E2 -24167.199} C_VEL
LIN {X 0,Y 181.803,Z 499.477,A -85,B 0,C 180,E1 -24168.921,E2 -24168.921} C_VEL
LIN {X 0,Y 176.643,Z 508.763,A -85,B 0,C 180,E1 -24171.202,E2 -24171.202} C_VEL
LIN {X 0,Y 170.953,Z 517.766,A -85,B 0,C 180,E1 -24174.143,E2 -24174.143} C_VEL
LIN {X 0,Y 165.638,Z 525.057,A -85,B 0,C 180,E1 -24177.254,E2 -24177.254} C_VEL
LIN {X 0,Y 161.804,Z 530.018,A -85,B 0,C 180,E1 -24180.037,E2 -24180.037} C_VEL
LIN {X 0,Y 157.927,Z 534.863,A -85,B 0,C 180,E1 -24183.58,E2 -24183.58} C_VEL
LIN {X 0,Y 154.462,Z 538.627,A -85,B 0,C 180,E1 -24187.252,E2 -24187.252} C_VEL
LIN {X 0,Y 151.634,Z 541.403,A -85,B 0,C 180,E1 -24191.073,E2 -24191.073} C_VEL
LIN {X 0,Y 149.173,Z 543.687,A -85,B 0,C 180,E1 -24196.379,E2 -24196.379} C_VEL
LIN {X 0,Y 148.809,Z 543.927,A -85,B 0,C 180,E1 -24197.531,E2 -24197.531} C_VEL
LIN {X 0,Y 147.596,Z 544.298,A -85,B 0,C 180,E1 -24199.762,E2 -24199.762} C_VEL
LIN {X 0,Y 144.226,Z 544.148,A -85,B 0,C 180,E1 -24203.424,E2 -24203.424} C_VEL
LIN {X 0,Y 141.711,Z 543.43,A -85,B 0,C 180,E1 -24206.452,E2 -24206.452} C_VEL
LIN {X 0,Y 140.779,Z 542.601,A -85,B 0,C 180,E1 -24208.817,E2 -24208.817} C_VEL
LIN {X 0,Y 140.764,Z 542.274,A -85,B 0,C 180,E1 -24209.616,E2 -24209.616} C_VEL
LIN {X 0,Y 140.659,Z 540.583,A -85,B 0,C 180,E1 -24212.868,E2 -24212.868} C_VEL
LIN {X 0,Y 140.795,Z 537.46,A -85,B 0,C 180,E1 -24217.173,E2 -24217.173} C_VEL
LIN {X 0,Y 141.367,Z 533.236,A -85,B 0,C 180,E1 -24221.474,E2 -24221.474} C_VEL
LIN {X 0,Y 142.748,Z 526.77,A -85,B 0,C 180,E1 -24226.449,E2 -24226.449} C_VEL
LIN {X 0,Y 144.822,Z 519.703,A -85,B 0,C 180,E1 -24230.604,E2 -24230.604} C_VEL
LIN {X 0,Y 146.973,Z 512.522,A -85,B 0,C 180,E1 -24233.957,E2 -24233.957} C_VEL
LIN {X 0,Y 148.367,Z 507.732,A -85,B 0,C 180,E1 -24235.839,E2 -24235.839} C_VEL
LIN {X 0,Y 151.138,Z 498.529,A -85,B 0,C 180,E1 -24238.849,E2 -24238.849} C_VEL
LIN {X 0,Y 153.686,Z 488.979,A -85,B 0,C 180,E1 -24241.348,E2 -24241.348} C_VEL
LIN {X 0,Y 156.817,Z 477.204,A -85,B 0,C 180,E1 -24243.688,E2 -24243.688} C_VEL
LIN {X 0,Y 159.218,Z 465.681,A -85,B 0,C 180,E1 -24245.409,E2 -24245.409} C_VEL
LIN {X 0,Y 161.302,Z 452.68,A -85,B 0,C 180,E1 -24246.809,E2 -24246.809} C_VEL
LIN {X 0,Y 162.757,Z 439.604,A -85,B 0,C 180,E1 -24247.728,E2 -24247.728} C_VEL
LIN {X 0,Y 165.164,Z 395.374,A -85,B 0,C 180,E1 -24249.534,E2 -24249.534} C_VEL
LIN {X 0,Y 163.604,Z 376.944,A -85,B 0,C 180,E1 -24250.861,E2 -24250.861} C_VEL
LIN {X 0,Y 158.193,Z 362.013,A -85,B 0,C 180,E1 -24253.033,E2 -24253.033} C_VEL
LIN {X 0,Y 152.4,Z 349.031,A -85,B 0,C 180,E1 -24255.429,E2 -24255.429} C_VEL
LIN {X 0,Y 148.247,Z 341.335,A -85,B 0,C 180,E1 -24257.216,E2 -24257.216} C_VEL
LIN {X 0,Y 146.04,Z 337.958,A -85,B 0,C 180,E1 -24258.18,E2 -24258.18} C_VEL
LIN {X 0,Y 145.15,Z 336.795,A -85,B 0,C 180,E1 -24258.568,E2 -24258.568} C_VEL
LIN {X 0,Y 143.519,Z 334.36,A -85,B 0,C 180,E1 -24259.319,E2 -24259.319} C_VEL
LIN {X 0,Y 143.071,Z 332.657,A -85,B 0,C 180,E1 -24259.659,E2 -24259.659} C_VEL
LIN {X 0,Y 143.096,Z 332.657,A -85,B 0,C 180,E1 -24263.887,E2 -24263.887} C_VEL
LIN {X 0,Y 143.191,Z 332.644,A -85,B 0,C 180,E1 -24267.323,E2 -24267.323} C_VEL
LIN {X 0,Y 143.197,Z 332.646,A -85,B 0,C 180,E1 -24272.066,E2 -24272.066} C_VEL
LIN {X 0,Y 143.236,Z 332.632,A -85,B 0,C 180,E1 -24278.798,E2 -24278.798} C_VEL
LIN {X 0,Y 143.268,Z 332.609,A -85,B 0,C 180,E1 -24282.882,E2 -24282.882} C_VEL
LIN {X 0,Y 143.543,Z 332.601,A -85,B 0,C 180,E1 -24288.705,E2 -24288.705} C_VEL
LIN {X 0,Y 143.617,Z 332.563,A -85,B 0,C 180,E1 -24291.557,E2 -24291.557} C_VEL
LIN {X 0,Y 144.183,Z 332.522,A -85,B 0,C 180,E1 -24299.999,E2 -24299.999} C_VEL
LIN {X 0,Y 143.633,Z 332.566,A -85,B 0,C 180,E1 -24308.44,E2 -24308.44} C_VEL
LIN {X 0,Y 143.509,Z 332.606,A -85,B 0,C 180,E1 -24311.619,E2 -24311.619} C_VEL
LIN {X 0,Y 143.276,Z 332.631,A -85,B 0,C 180,E1 -24317.116,E2 -24317.116} C_VEL
LIN {X 0,Y 143.275,Z 332.63,A -85,B 0,C 180,E1 -24321.242,E2 -24321.242} C_VEL
LIN {X 0,Y 143.196,Z 332.638,A -85,B 0,C 180,E1 -24327.933,E2 -24327.933} C_VEL
LIN {X 0,Y 143.151,Z 332.644,A -85,B 0,C 180,E1 -24333.418,E2 -24333.418} C_VEL
LIN {X 0,Y 143.063,Z 332.652,A -85,B 0,C 180,E1 -24339.689,E2 -24339.689} C_VEL
LIN {X 0,Y 143.058,Z 332.661,A -85,B 0,C 180,E1 -24343.454,E2 -24343.454} C_VEL
LIN {X 0,Y 143.045,Z 332.663,A -85,B 0,C 180,E1 -24347.473,E2 -24347.473} C_VEL
LIN {X 0,Y 143.08,Z 332.659,A -85,B 0,C 180,E1 -24351.804,E2 -24351.804} C_VEL
LIN {X 0,Y 143.186,Z 332.844,A -85,B 0,C 180,E1 -24356.071,E2 -24356.071} C_VEL
LIN {X 0,Y 144.234,Z 335.629,A -85,B 0,C 180,E1 -24356.642,E2 -24356.642} C_VEL
LIN {X 0,Y 146.146,Z 337.876,A -85,B 0,C 180,E1 -24357.466,E2 -24357.466} C_VEL
LIN {X 0,Y 154.056,Z 350.764,A -85,B 0,C 180,E1 -24360.776,E2 -24360.776} C_VEL
LIN {X 0,Y 160.48,Z 362.752,A -85,B 0,C 180,E1 -24363.214,E2 -24363.214} C_VEL
LIN {X 0,Y 166.051,Z 375.17,A -85,B 0,C 180,E1 -24365.227,E2 -24365.227} C_VEL
LIN {X 0,Y 163.72,Z 417.703,A -85,B 0,C 180,E1 -24366.904,E2 -24366.904} C_VEL
LIN {X 0,Y 162.526,Z 434.126,A -85,B 0,C 180,E1 -24367.68,E2 -24367.68} C_VEL
LIN {X 0,Y 161.052,Z 446.573,A -85,B 0,C 180,E1 -24368.728,E2 -24368.728} C_VEL
LIN {X 0,Y 159.046,Z 459.205,A -85,B 0,C 180,E1 -24370.306,E2 -24370.306} C_VEL
LIN {X 0,Y 156.411,Z 471.385,A -85,B 0,C 180,E1 -24372.34,E2 -24372.34} C_VEL
LIN {X 0,Y 153.869,Z 482.156,A -85,B 0,C 180,E1 -24374.77,E2 -24374.77} C_VEL
LIN {X 0,Y 151.062,Z 491.91,A -85,B 0,C 180,E1 -24377.535,E2 -24377.535} C_VEL
LIN {X 0,Y 148.047,Z 501.792,A -85,B 0,C 180,E1 -24381.121,E2 -24381.121} C_VEL
LIN {X 0,Y 145.369,Z 510.327,A -85,B 0,C 180,E1 -24385.143,E2 -24385.143} C_VEL
LIN {X 0,Y 143.354,Z 517.174,A -85,B 0,C 180,E1 -24389.294,E2 -24389.294} C_VEL
LIN {X 0,Y 141.759,Z 523.467,A -85,B 0,C 180,E1 -24394.26,E2 -24394.26} C_VEL
LIN {X 0,Y 140.799,Z 527.581,A -85,B 0,C 180,E1 -24398.608,E2 -24398.608} C_VEL
LIN {X 0,Y 140.423,Z 529.706,A -85,B 0,C 180,E1 -24401.544,E2 -24401.544} C_VEL
LIN {X 0,Y 140.303,Z 531.401,A -85,B 0,C 180,E1 -24404.5,E2 -24404.5} C_VEL
LIN {X 0,Y 140.499,Z 532.888,A -85,B 0,C 180,E1 -24408.121,E2 -24408.121} C_VEL
LIN {X 0,Y 141.389,Z 533.909,A -85,B 0,C 180,E1 -24413.427,E2 -24413.427} C_VEL
LIN {X 0,Y 142.842,Z 533.758,A -85,B 0,C 180,E1 -24417.673,E2 -24417.673} C_VEL
LIN {X 0,Y 145.082,Z 532.588,A -85,B 0,C 180,E1 -24422.193,E2 -24422.193} C_VEL
LIN {X 0,Y 147.728,Z 530.691,A -85,B 0,C 180,E1 -24426.026,E2 -24426.026} C_VEL
LIN {X 0,Y 151.646,Z 527.241,A -85,B 0,C 180,E1 -24430.447,E2 -24430.447} C_VEL
LIN {X 0,Y 155.958,Z 522.918,A -85,B 0,C 180,E1 -24434.258,E2 -24434.258} C_VEL
LIN {X 0,Y 160.936,Z 517.224,A -85,B 0,C 180,E1 -24437.928,E2 -24437.928} C_VEL
LIN {X 0,Y 166.505,Z 510.077,A -85,B 0,C 180,E1 -24441.333,E2 -24441.333} C_VEL
LIN {X 0,Y 171.507,Z 502.673,A -85,B 0,C 180,E1 -24444.022,E2 -24444.022} C_VEL
LIN {X 0,Y 176.943,Z 493.621,A -85,B 0,C 180,E1 -24446.515,E2 -24446.515} C_VEL
LIN {X 0,Y 182.036,Z 483.588,A -85,B 0,C 180,E1 -24448.663,E2 -24448.663} C_VEL
LIN {X 0,Y 186.71,Z 472.642,A -85,B 0,C 180,E1 -24450.452,E2 -24450.452} C_VEL
LIN {X 0,Y 190.525,Z 461.461,A -85,B 0,C 180,E1 -24451.844,E2 -24451.844} C_VEL
LIN {X 0,Y 193.747,Z 449.382,A -85,B 0,C 180,E1 -24452.949,E2 -24452.949} C_VEL
LIN {X 0,Y 196.235,Z 436.413,A -85,B 0,C 180,E1 -24453.771,E2 -24453.771} C_VEL
LIN {X 0,Y 197.838,Z 422.302,A -85,B 0,C 180,E1 -24454.293,E2 -24454.293} C_VEL
LIN {X 0,Y 199.24,Z 404.878,A -85,B 0,C 180,E1 -24454.819,E2 -24454.819} C_VEL
LIN {X 0,Y 195.642,Z 397.79,A -85,B 0,C 180,E1 -24456.939,E2 -24456.939} C_VEL
LIN {X 0,Y 190.107,Z 388.236,A -85,B 0,C 180,E1 -24460.567,E2 -24460.567} C_VEL
LIN {X 0,Y 185.588,Z 381.195,A -85,B 0,C 180,E1 -24464.065,E2 -24464.065} C_VEL
LIN {X 0,Y 182.568,Z 376.737,A -85,B 0,C 180,E1 -24466.791,E2 -24466.791} C_VEL
LIN {X 0,Y 180.008,Z 372.94,A -85,B 0,C 180,E1 -24469.485,E2 -24469.485} C_VEL
LIN {X 0,Y 177.468,Z 369.556,A -85,B 0,C 180,E1 -24472.641,E2 -24472.641} C_VEL
LIN {X 0,Y 176.944,Z 368.349,A -85,B 0,C 180,E1 -24473.494,E2 -24473.494} C_VEL
LIN {X 0,Y 174.399,Z 365.696,A -85,B 0,C 180,E1 -24478.016,E2 -24478.016} C_VEL
LIN {X 0,Y 173.521,Z 363.055,A -85,B 0,C 180,E1 -24480.829,E2 -24480.829} C_VEL
LIN {X 0,Y 172.522,Z 362.849,A -85,B 0,C 180,E1 -24489.379,E2 -24489.379} C_VEL
LIN {X 0,Y 173.374,Z 363.355,A -85,B 0,C 180,E1 -24493.392,E2 -24493.392} C_VEL
LIN {X 0,Y 174.981,Z 366.935,A -85,B 0,C 180,E1 -24497.882,E2 -24497.882} C_VEL
LIN {X 0,Y 177.005,Z 368.946,A -85,B 0,C 180,E1 -24501.229,E2 -24501.229} C_VEL
LIN {X 0,Y 180.901,Z 375.348,A -85,B 0,C 180,E1 -24506.169,E2 -24506.169} C_VEL
LIN {X 0,Y 184.023,Z 380.811,A -85,B 0,C 180,E1 -24509.306,E2 -24509.306} C_VEL
LIN {X 0,Y 187.038,Z 386.489,A -85,B 0,C 180,E1 -24511.939,E2 -24511.939} C_VEL
LIN {X 0,Y 190.94,Z 394.243,A -85,B 0,C 180,E1 -24514.925,E2 -24514.925} C_VEL
LIN {X 0,Y 194.914,Z 402.992,A -85,B 0,C 180,E1 -24517.612,E2 -24517.612} C_VEL
LIN {X 0,Y 198.64,Z 412.707,A -85,B 0,C 180,E1 -24519.966,E2 -24519.966} C_VEL
LIN {X 0,Y 196.194,Z 440.653,A -85,B 0,C 180,E1 -24520.86,E2 -24520.86} C_VEL
LIN {X 0,Y 193.859,Z 454.01,A -85,B 0,C 180,E1 -24521.547,E2 -24521.547} C_VEL
LIN {X 0,Y 190.683,Z 466.487,A -85,B 0,C 180,E1 -24522.517,E2 -24522.517} C_VEL
LIN {X 0,Y 186.337,Z 478.961,A -85,B 0,C 180,E1 -24523.841,E2 -24523.841} C_VEL
LIN {X 0,Y 181.623,Z 490.09,A -85,B 0,C 180,E1 -24525.469,E2 -24525.469} C_VEL
LIN {X 0,Y 176.553,Z 500.143,A -85,B 0,C 180,E1 -24527.418,E2 -24527.418} C_VEL
LIN {X 0,Y 171.198,Z 509.235,A -85,B 0,C 180,E1 -24529.722,E2 -24529.722} C_VEL
LIN {X 0,Y 165.253,Z 518.116,A -85,B 0,C 180,E1 -24532.702,E2 -24532.702} C_VEL
LIN {X 0,Y 159.71,Z 525.3,A -85,B 0,C 180,E1 -24535.876,E2 -24535.876} C_VEL
LIN {X 0,Y 155.694,Z 530.164,A -85,B 0,C 180,E1 -24538.733,E2 -24538.733} C_VEL
LIN {X 0,Y 151.58,Z 534.921,A -85,B 0,C 180,E1 -24542.382,E2 -24542.382} C_VEL
LIN {X 0,Y 147.904,Z 538.6,A -85,B 0,C 180,E1 -24546.183,E2 -24546.183} C_VEL
LIN {X 0,Y 144.932,Z 541.298,A -85,B 0,C 180,E1 -24550.162,E2 -24550.162} C_VEL
LIN {X 0,Y 142.249,Z 543.506,A -85,B 0,C 180,E1 -24555.703,E2 -24555.703} C_VEL
LIN {X 0,Y 140.9,Z 544.109,A -85,B 0,C 180,E1 -24561.398,E2 -24561.398} C_VEL
LIN {X 0,Y 140.682,Z 543.841,A -85,B 0,C 180,E1 -24564.27,E2 -24564.27} C_VEL
LIN {X 0,Y 140.667,Z 542.986,A -85,B 0,C 180,E1 -24567.784,E2 -24567.784} C_VEL
LIN {X 0,Y 140.764,Z 542.274,A -85,B 0,C 180,E1 -24569.616,E2 -24569.616} C_VEL
LIN {X 0,Y 140.553,Z 541.56,A -85,B 0,C 180,E1 -24571.184,E2 -24571.184} C_VEL
LIN {X 0,Y 139.789,Z 540.68,A -85,B 0,C 180,E1 -24572.719,E2 -24572.719} C_VEL
LIN {X 0,Y 137.401,Z 538.524,A -85,B 0,C 180,E1 -24575.727,E2 -24575.727} C_VEL
LIN {X 0,Y 135.058,Z 535.918,A -85,B 0,C 180,E1 -24578.786,E2 -24578.786} C_VEL
LIN {X 0,Y 134.27,Z 533.646,A -85,B 0,C 180,E1 -24581.131,E2 -24581.131} C_VEL
LIN {X 0,Y 134.327,Z 532.792,A -85,B 0,C 180,E1 -24581.914,E2 -24581.914} C_VEL
LIN {X 0,Y 135.604,Z 527.082,A -85,B 0,C 180,E1 -24586.566,E2 -24586.566} C_VEL
LIN {X 0,Y 137.76,Z 520.165,A -85,B 0,C 180,E1 -24590.927,E2 -24590.927} C_VEL
LIN {X 0,Y 140.283,Z 511.991,A -85,B 0,C 180,E1 -24594.957,E2 -24594.957} C_VEL
LIN {X 0,Y 142.08,Z 506.503,A -85,B 0,C 180,E1 -24597.153,E2 -24597.153} C_VEL
LIN {X 0,Y 144.58,Z 498.396,A -85,B 0,C 180,E1 -24599.889,E2 -24599.889} C_VEL
LIN {X 0,Y 147.241,Z 488.866,A -85,B 0,C 180,E1 -24602.482,E2 -24602.482} C_VEL
LIN {X 0,Y 150.063,Z 478.721,A -85,B 0,C 180,E1 -24604.605,E2 -24604.605} C_VEL
LIN {X 0,Y 152.768,Z 466.772,A -85,B 0,C 180,E1 -24606.53,E2 -24606.53} C_VEL
LIN {X 0,Y 154.932,Z 454.273,A -85,B 0,C 180,E1 -24607.972,E2 -24607.972} C_VEL
LIN {X 0,Y 156.651,Z 440.614,A -85,B 0,C 180,E1 -24608.997,E2 -24608.997} C_VEL
LIN {X 0,Y 159.201,Z 397.147,A -85,B 0,C 180,E1 -24610.837,E2 -24610.837} C_VEL
LIN {X 0,Y 157.87,Z 379.184,A -85,B 0,C 180,E1 -24612.157,E2 -24612.157} C_VEL
LIN {X 0,Y 152.75,Z 364.884,A -85,B 0,C 180,E1 -24614.376,E2 -24614.376} C_VEL
LIN {X 0,Y 147.509,Z 352.986,A -85,B 0,C 180,E1 -24616.714,E2 -24616.714} C_VEL
LIN {X 0,Y 144.014,Z 346.3,A -85,B 0,C 180,E1 -24618.335,E2 -24618.335} C_VEL
LIN {X 0,Y 139.29,Z 339.177,A -85,B 0,C 180,E1 -24620.591,E2 -24620.591} C_VEL
LIN {X 0,Y 138.349,Z 337.94,A -85,B 0,C 180,E1 -24621.057,E2 -24621.057} C_VEL
LIN {X 0,Y 136.682,Z 335.734,A -85,B 0,C 180,E1 -24621.9,E2 -24621.9} C_VEL
LIN {X 0,Y 136.05,Z 333.53,A -85,B 0,C 180,E1 -24622.395,E2 -24622.395} C_VEL
LIN {X 0,Y 136.064,Z 333.527,A -85,B 0,C 180,E1 -24625.741,E2 -24625.741} C_VEL
LIN {X 0,Y 136.153,Z 333.524,A -85,B 0,C 180,E1 -24632.317,E2 -24632.317} C_VEL
LIN {X 0,Y 136.202,Z 333.508,A -85,B 0,C 180,E1 -24638.825,E2 -24638.825} C_VEL
LIN {X 0,Y 136.239,Z 333.503,A -85,B 0,C 180,E1 -24645.052,E2 -24645.052} C_VEL
LIN {X 0,Y 136.435,Z 333.487,A -85,B 0,C 180,E1 -24648.178,E2 -24648.178} C_VEL
LIN {X 0,Y 136.546,Z 333.446,A -85,B 0,C 180,E1 -24651.117,E2 -24651.117} C_VEL
LIN {X 0,Y 137.14,Z 333.399,A -85,B 0,C 180,E1 -24659.999,E2 -24659.999} C_VEL
LIN {X 0,Y 136.558,Z 333.451,A -85,B 0,C 180,E1 -24668.881,E2 -24668.881} C_VEL
LIN {X 0,Y 136.424,Z 333.489,A -85,B 0,C 180,E1 -24671.891,E2 -24671.891} C_VEL
LIN {X 0,Y 136.196,Z 333.518,A -85,B 0,C 180,E1 -24678.035,E2 -24678.035} C_VEL
LIN {X 0,Y 136.198,Z 333.509,A -85,B 0,C 180,E1 -24681.737,E2 -24681.737} C_VEL
LIN {X 0,Y 136.106,Z 333.518,A -85,B 0,C 180,E1 -24688.612,E2 -24688.612} C_VEL
LIN {X 0,Y 136.05,Z 333.524,A -85,B 0,C 180,E1 -24694.626,E2 -24694.626} C_VEL
LIN {X 0,Y 136.036,Z 333.529,A -85,B 0,C 180,E1 -24699.194,E2 -24699.194} C_VEL
LIN {X 0,Y 135.999,Z 333.539,A -85,B 0,C 180,E1 -24703.652,E2 -24703.652} C_VEL
LIN {X 0,Y 135.989,Z 333.543,A -85,B 0,C 180,E1 -24707.785,E2 -24707.785} C_VEL
LIN {X 0,Y 136.045,Z 333.667,A -85,B 0,C 180,E1 -24713.281,E2 -24713.281} C_VEL
LIN {X 0,Y 137.082,Z 336.437,A -85,B 0,C 180,E1 -24713.927,E2 -24713.927} C_VEL
LIN {X 0,Y 139.349,Z 339.112,A -85,B 0,C 180,E1 -24715.04,E2 -24715.04} C_VEL
LIN {X 0,Y 141.388,Z 342.244,A -85,B 0,C 180,E1 -24716.045,E2 -24716.045} C_VEL
LIN {X 0,Y 146.724,Z 350.703,A -85,B 0,C 180,E1 -24718.491,E2 -24718.491} C_VEL
LIN {X 0,Y 152.526,Z 360.876,A -85,B 0,C 180,E1 -24720.928,E2 -24720.928} C_VEL
LIN {X 0,Y 158.914,Z 374.312,A -85,B 0,C 180,E1 -24723.449,E2 -24723.449} C_VEL
LIN {X 0,Y 160.133,Z 377.263,A -85,B 0,C 180,E1 -24723.92,E2 -24723.92} C_VEL
LIN {X 0,Y 156.845,Z 430.995,A -85,B 0,C 180,E1 -24726.142,E2 -24726.142} C_VEL
LIN {X 0,Y 155.253,Z 444.563,A -85,B 0,C 180,E1 -24727.19,E2 -24727.19} C_VEL
LIN {X 0,Y 153.372,Z 456.885,A -85,B 0,C 180,E1 -24728.667,E2 -24728.667} C_VEL
LIN {X 0,Y 150.772,Z 468.807,A -85,B 0,C 180,E1 -24730.598,E2 -24730.598} C_VEL
LIN {X 0,Y 147.958,Z 480.211,A -85,B 0,C 180,E1 -24733.082,E2 -24733.082} C_VEL
LIN {X 0,Y 144.973,Z 490.52,A -85,B 0,C 180,E1 -24735.968,E2 -24735.968} C_VEL
LIN {X 0,Y 142.078,Z 499.766,A -85,B 0,C 180,E1 -24739.306,E2 -24739.306} C_VEL
LIN {X 0,Y 139.076,Z 508.778,A -85,B 0,C 180,E1 -24743.467,E2 -24743.467} C_VEL
LIN {X 0,Y 136.783,Z 516.016,A -85,B 0,C 180,E1 -24747.787,E2 -24747.787} C_VEL
LIN {X 0,Y 135.393,Z 520.897,A -85,B 0,C 180,E1 -24751.483,E2 -24751.483} C_VEL
LIN {X 0,Y 134.228,Z 525.647,A -85,B 0,C 180,E1 -24756.006,E2 -24756.006} C_VEL
LIN {X 0,Y 133.406,Z 529.295,A -85,B 0,C 180,E1 -24760.621,E2 -24760.621} C_VEL
LIN {X 0,Y 133.234,Z 531.899,A -85,B 0,C 180,E1 -24765.288,E2 -24765.288} C_VEL
LIN {X 0,Y 133.455,Z 533.141,A -85,B 0,C 180,E1 -24768.575,E2 -24768.575} C_VEL
LIN {X 0,Y 134.602,Z 534.209,A -85,B 0,C 180,E1 -24774.684,E2 -24774.684} C_VEL
LIN {X 0,Y 136.012,Z 534.046,A -85,B 0,C 180,E1 -24778.548,E2 -24778.548} C_VEL
LIN {X 0,Y 138.804,Z 532.686,A -85,B 0,C 180,E1 -24783.84,E2 -24783.84} C_VEL
LIN {X 0,Y 141.323,Z 531.016,A -85,B 0,C 180,E1 -24787.281,E2 -24787.281} C_VEL
LIN {X 0,Y 146.032,Z 527.123,A -85,B 0,C 180,E1 -24792.353,E2 -24792.353} C_VEL
LIN {X 0,Y 150.566,Z 522.81,A -85,B 0,C 180,E1 -24796.144,E2 -24796.144} C_VEL
LIN {X 0,Y 156.035,Z 516.86,A -85,B 0,C 180,E1 -24799.962,E2 -24799.962} C_VEL
LIN {X 0,Y 161.922,Z 509.497,A -85,B 0,C 180,E1 -24803.407,E2 -24803.407} C_VEL
LIN {X 0,Y 167.259,Z 501.919,A -85,B 0,C 180,E1 -24806.078,E2 -24806.078} C_VEL
LIN {X 0,Y 172.969,Z 492.665,A -85,B 0,C 180,E1 -24808.56,E2 -24808.56} C_VEL
LIN {X 0,Y 178.282,Z 482.365,A -85,B 0,C 180,E1 -24810.705,E2 -24810.705} C_VEL
LIN {X 0,Y 182.975,Z 471.45,A -85,B 0,C 180,E1 -24812.4,E2 -24812.4} C_VEL
LIN {X 0,Y 187.281,Z 458.661,A -85,B 0,C 180,E1 -24813.92,E2 -24813.92} C_VEL
LIN {X 0,Y 190.476,Z 446.274,A -85,B 0,C 180,E1 -24814.939,E2 -24814.939} C_VEL
LIN {X 0,Y 192.814,Z 432.95,A -85,B 0,C 180,E1 -24815.668,E2 -24815.668} C_VEL
LIN {X 0,Y 195.128,Z 407.89,A -85,B 0,C 180,E1 -24816.478,E2 -24816.478} C_VEL
LIN {X 0,Y 190.92,Z 399.93,A -85,B 0,C 180,E1 -24819.179,E2 -24819.179} C_VEL
LIN {X 0,Y 186.711,Z 392.53,A -85,B 0,C 180,E1 -24822.273,E2 -24822.273} C_VEL
LIN {X 0,Y 182.939,Z 386.572,A -85,B 0,C 180,E1 -24825.46,E2 -24825.46} C_VEL
LIN {X 0,Y 180.807,Z 383.225,A -85,B 0,C 180,E1 -24827.534,E2 -24827.534} C_VEL
LIN {X 0,Y 178.37,Z 379.486,A -85,B 0,C 180,E1 -24830.248,E2 -24830.248} C_VEL
LIN {X 0,Y 175.983,Z 376.026,A -85,B 0,C 180,E1 -24833.458,E2 -24833.458} C_VEL
LIN {X 0,Y 175.51,Z 375.099,A -85,B 0,C 180,E1 -24834.255,E2 -24834.255} C_VEL
LIN {X 0,Y 173.18,Z 372.284,A -85,B 0,C 180,E1 -24838.82,E2 -24838.82} C_VEL
LIN {X 0,Y 172.542,Z 370.096,A -85,B 0,C 180,E1 -24841.111,E2 -24841.111} C_VEL
LIN {X 0,Y 171.651,Z 369.898,A -85,B 0,C 180,E1 -24849.427,E2 -24849.427} C_VEL
LIN {X 0,Y 172.39,Z 370.425,A -85,B 0,C 180,E1 -24853.086,E2 -24853.086} C_VEL
LIN {X 0,Y 174.261,Z 374.318,A -85,B 0,C 180,E1 -24858.246,E2 -24858.246} C_VEL
LIN {X 0,Y 175.625,Z 375.61,A -85,B 0,C 180,E1 -24860.538,E2 -24860.538} C_VEL
LIN {X 0,Y 179.138,Z 381.732,A -85,B 0,C 180,E1 -24865.325,E2 -24865.325} C_VEL
LIN {X 0,Y 181.933,Z 386.867,A -85,B 0,C 180,E1 -24868.328,E2 -24868.328} C_VEL
LIN {X 0,Y 185.44,Z 393.773,A -85,B 0,C 180,E1 -24871.55,E2 -24871.55} C_VEL
LIN {X 0,Y 189.501,Z 402.514,A -85,B 0,C 180,E1 -24874.782,E2 -24874.782} C_VEL
LIN {X 0,Y 193.114,Z 411.327,A -85,B 0,C 180,E1 -24877.33,E2 -24877.33} C_VEL
LIN {X 0,Y 194.538,Z 415.25,A -85,B 0,C 180,E1 -24878.291,E2 -24878.291} C_VEL
LIN {X 0,Y 192.217,Z 440.713,A -85,B 0,C 180,E1 -24879.123,E2 -24879.123} C_VEL
LIN {X 0,Y 189.798,Z 454.054,A -85,B 0,C 180,E1 -24879.811,E2 -24879.811} C_VEL
LIN {X 0,Y 186.532,Z 466.39,A -85,B 0,C 180,E1 -24880.768,E2 -24880.768} C_VEL
LIN {X 0,Y 182.164,Z 478.552,A -85,B 0,C 180,E1 -24882.046,E2 -24882.046} C_VEL
LIN {X 0,Y 177.266,Z 489.71,A -85,B 0,C 180,E1 -24883.657,E2 -24883.657} C_VEL
LIN {X 0,Y 171.978,Z 499.793,A -85,B 0,C 180,E1 -24885.593,E2 -24885.593} C_VEL
LIN {X 0,Y 165.877,Z 509.707,A -85,B 0,C 180,E1 -24888.146,E2 -24888.146} C_VEL
LIN {X 0,Y 159.678,Z 518.466,A -85,B 0,C 180,E1 -24891.162,E2 -24891.162} C_VEL
LIN {X 0,Y 153.891,Z 525.516,A -85,B 0,C 180,E1 -24894.394,E2 -24894.394} C_VEL
LIN {X 0,Y 149.65,Z 530.311,A -85,B 0,C 180,E1 -24897.317,E2 -24897.317} C_VEL
LIN {X 0,Y 145.301,Z 534.98,A -85,B 0,C 180,E1 -24901.079,E2 -24901.079} C_VEL
LIN {X 0,Y 141.406,Z 538.577,A -85,B 0,C 180,E1 -24905.015,E2 -24905.015} C_VEL
LIN {X 0,Y 138.247,Z 541.197,A -85,B 0,C 180,E1 -24909.159,E2 -24909.159} C_VEL
LIN {X 0,Y 136.559,Z 542.454,A -85,B 0,C 180,E1 -24912.019,E2 -24912.019} C_VEL
LIN {X 0,Y 135.355,Z 543.307,A -85,B 0,C 180,E1 -24914.958,E2 -24914.958} C_VEL
LIN {X 0,Y 133.863,Z 543.825,A -85,B 0,C 180,E1 -24920.943,E2 -24920.943} C_VEL
LIN {X 0,Y 133.615,Z 543.522,A -85,B 0,C 180,E1 -24923.966,E2 -24923.966} C_VEL
LIN {X 0,Y 133.612,Z 542.466,A -85,B 0,C 180,E1 -24928.042,E2 -24928.042} C_VEL
LIN {X 0,Y 133.603,Z 540.81,A -85,B 0,C 180,E1 -24931.852,E2 -24931.852} C_VEL
LIN {X 0,Y 133.632,Z 538.121,A -85,B 0,C 180,E1 -24936.042,E2 -24936.042} C_VEL
LIN {X 0,Y 134.098,Z 534.194,A -85,B 0,C 180,E1 -24940.574,E2 -24940.574} C_VEL
LIN {X 0,Y 134.327,Z 532.792,A -85,B 0,C 180,E1 -24941.914,E2 -24941.914} C_VEL
LIN {X 0,Y 134.195,Z 530.242,A -85,B 0,C 180,E1 -24944.19,E2 -24944.19} C_VEL
LIN {X 0,Y 132.551,Z 525.513,A -85,B 0,C 180,E1 -24947.876,E2 -24947.876} C_VEL
LIN {X 0,Y 131.364,Z 520.187,A -85,B 0,C 180,E1 -24951.479,E2 -24951.479} C_VEL
LIN {X 0,Y 131.944,Z 516.604,A -85,B 0,C 180,E1 -24953.531,E2 -24953.531} C_VEL
LIN {X 0,Y 133.615,Z 511.434,A -85,B 0,C 180,E1 -24956.057,E2 -24956.057} C_VEL
LIN {X 0,Y 137.14,Z 501.372,A -85,B 0,C 180,E1 -24959.982,E2 -24959.982} C_VEL
LIN {X 0,Y 140.226,Z 491.337,A -85,B 0,C 180,E1 -24963.032,E2 -24963.032} C_VEL
LIN {X 0,Y 143.355,Z 480.185,A -85,B 0,C 180,E1 -24965.608,E2 -24965.608} C_VEL
LIN {X 0,Y 145.92,Z 469.684,A -85,B 0,C 180,E1 -24967.454,E2 -24967.454} C_VEL
LIN {X 0,Y 148.226,Z 458.424,A -85,B 0,C 180,E1 -24968.925,E2 -24968.925} C_VEL
LIN {X 0,Y 150.094,Z 445.92,A -85,B 0,C 180,E1 -24970.083,E2 -24970.083} C_VEL
LIN {X 0,Y 151.259,Z 433.295,A -85,B 0,C 180,E1 -24970.806,E2 -24970.806} C_VEL
LIN {X 0,Y 153.338,Z 396.863,A -85,B 0,C 180,E1 -24972.348,E2 -24972.348} C_VEL
LIN {X 0,Y 152.14,Z 381.198,A -85,B 0,C 180,E1 -24973.587,E2 -24973.587} C_VEL
LIN {X 0,Y 147.435,Z 367.845,A -85,B 0,C 180,E1 -24975.8,E2 -24975.8} C_VEL
LIN {X 0,Y 142.613,Z 356.729,A -85,B 0,C 180,E1 -24978.13,E2 -24978.13} C_VEL
LIN {X 0,Y 139.693,Z 351.12,A -85,B 0,C 180,E1 -24979.587,E2 -24979.587} C_VEL
LIN {X 0,Y 134.669,Z 343.473,A -85,B 0,C 180,E1 -24982.178,E2 -24982.178} C_VEL
LIN {X 0,Y 132.388,Z 340.064,A -85,B 0,C 180,E1 -24983.447,E2 -24983.447} C_VEL
LIN {X 0,Y 131.722,Z 339.146,A -85,B 0,C 180,E1 -24983.825,E2 -24983.825} C_VEL
LIN {X 0,Y 129.862,Z 337.031,A -85,B 0,C 180,E1 -24984.881,E2 -24984.881} C_VEL
LIN {X 0,Y 129.017,Z 334.405,A -85,B 0,C 180,E1 -24985.568,E2 -24985.568} C_VEL
LIN {X 0,Y 129.026,Z 334.405,A -85,B 0,C 180,E1 -24990.644,E2 -24990.644} C_VEL
LIN {X 0,Y 129.032,Z 334.412,A -85,B 0,C 180,E1 -24994.167,E2 -24994.167} C_VEL
LIN {X 0,Y 129.082,Z 334.403,A -85,B 0,C 180,E1 -24997.767,E2 -24997.767} C_VEL
LIN {X 0,Y 129.16,Z 334.374,A -85,B 0,C 180,E1 -25004.212,E2 -25004.212} C_VEL
LIN {X 0,Y 129.354,Z 334.37,A -85,B 0,C 180,E1 -25007.97,E2 -25007.97} C_VEL
LIN {X 0,Y 129.471,Z 334.331,A -85,B 0,C 180,E1 -25010.627,E2 -25010.627} C_VEL
LIN {X 0,Y 130.095,Z 334.277,A -85,B 0,C 180,E1 -25019.999,E2 -25019.999} C_VEL
LIN {X 0,Y 129.48,Z 334.336,A -85,B 0,C 180,E1 -25029.371,E2 -25029.371} C_VEL
LIN {X 0,Y 129.308,Z 334.378,A -85,B 0,C 180,E1 -25032.556,E2 -25032.556} C_VEL
LIN {X 0,Y 129.123,Z 334.401,A -85,B 0,C 180,E1 -25039.06,E2 -25039.06} C_VEL
LIN {X 0,Y 129.115,Z 334.39,A -85,B 0,C 180,E1 -25042.397,E2 -25042.397} C_VEL
LIN {X 0,Y 129.034,Z 334.41,A -85,B 0,C 180,E1 -25045.831,E2 -25045.831} C_VEL
LIN {X 0,Y 129.024,Z 334.4,A -85,B 0,C 180,E1 -25049.355,E2 -25049.355} C_VEL
LIN {X 0,Y 128.966,Z 334.406,A -85,B 0,C 180,E1 -25055.165,E2 -25055.165} C_VEL
LIN {X 0,Y 128.937,Z 334.41,A -85,B 0,C 180,E1 -25060.85,E2 -25060.85} C_VEL
LIN {X 0,Y 128.921,Z 334.415,A -85,B 0,C 180,E1 -25065.127,E2 -25065.127} C_VEL
LIN {X 0,Y 128.949,Z 334.413,A -85,B 0,C 180,E1 -25069.997,E2 -25069.997} C_VEL
LIN {X 0,Y 129.932,Z 337.14,A -85,B 0,C 180,E1 -25070.765,E2 -25070.765} C_VEL
LIN {X 0,Y 132.348,Z 339.93,A -85,B 0,C 180,E1 -25072.125,E2 -25072.125} C_VEL
LIN {X 0,Y 134.473,Z 343.223,A -85,B 0,C 180,E1 -25073.324,E2 -25073.324} C_VEL
LIN {X 0,Y 135.936,Z 345.305,A -85,B 0,C 180,E1 -25074.104,E2 -25074.104} C_VEL
LIN {X 0,Y 139.931,Z 351.336,A -85,B 0,C 180,E1 -25076.126,E2 -25076.126} C_VEL
LIN {X 0,Y 146.597,Z 362.84,A -85,B 0,C 180,E1 -25079.223,E2 -25079.223} C_VEL
LIN {X 0,Y 153.194,Z 376.639,A -85,B 0,C 180,E1 -25082.049,E2 -25082.049} C_VEL
LIN {X 0,Y 154.225,Z 379.159,A -85,B 0,C 180,E1 -25082.481,E2 -25082.481} C_VEL
LIN {X 0,Y 150.94,Z 431.132,A -85,B 0,C 180,E1 -25084.693,E2 -25084.693} C_VEL
LIN {X 0,Y 149.261,Z 444.695,A -85,B 0,C 180,E1 -25085.758,E2 -25085.758} C_VEL
LIN {X 0,Y 147.198,Z 457.562,A -85,B 0,C 180,E1 -25087.356,E2 -25087.356} C_VEL
LIN {X 0,Y 144.474,Z 469.394,A -85,B 0,C 180,E1 -25089.345,E2 -25089.345} C_VEL
LIN {X 0,Y 141.521,Z 480.74,A -85,B 0,C 180,E1 -25091.914,E2 -25091.914} C_VEL
LIN {X 0,Y 138.554,Z 490.494,A -85,B 0,C 180,E1 -25094.747,E2 -25094.747} C_VEL
LIN {X 0,Y 135.628,Z 499.378,A -85,B 0,C 180,E1 -25098.033,E2 -25098.033} C_VEL
LIN {X 0,Y 132.416,Z 508.499,A -85,B 0,C 180,E1 -25102.371,E2 -25102.371} C_VEL
LIN {X 0,Y 129.946,Z 515.842,A -85,B 0,C 180,E1 -25106.895,E2 -25106.895} C_VEL
LIN {X 0,Y 128.204,Z 521.708,A -85,B 0,C 180,E1 -25111.566,E2 -25111.566} C_VEL
LIN {X 0,Y 127.033,Z 526.333,A -85,B 0,C 180,E1 -25116.348,E2 -25116.348} C_VEL
LIN {X 0,Y 126.242,Z 529.875,A -85,B 0,C 180,E1 -25121.231,E2 -25121.231} C_VEL
LIN {X 0,Y 126.15,Z 532.388,A -85,B 0,C 180,E1 -25126.169,E2 -25126.169} C_VEL
LIN {X 0,Y 126.45,Z 533.497,A -85,B 0,C 180,E1 -25129.475,E2 -25129.475} C_VEL
LIN {X 0,Y 126.984,Z 534.206,A -85,B 0,C 180,E1 -25132.789,E2 -25132.789} C_VEL
LIN {X 0,Y 127.907,Z 534.51,A -85,B 0,C 180,E1 -25136.071,E2 -25136.071} C_VEL
LIN {X 0,Y 129.224,Z 534.332,A -85,B 0,C 180,E1 -25139.522,E2 -25139.522} C_VEL
LIN {X 0,Y 132.668,Z 532.784,A -85,B 0,C 180,E1 -25145.636,E2 -25145.636} C_VEL
LIN {X 0,Y 134.995,Z 531.339,A -85,B 0,C 180,E1 -25148.656,E2 -25148.656} C_VEL
LIN {X 0,Y 139.08,Z 528.279,A -85,B 0,C 180,E1 -25153.008,E2 -25153.008} C_VEL
LIN {X 0,Y 143.904,Z 524.07,A -85,B 0,C 180,E1 -25157.095,E2 -25157.095} C_VEL
LIN {X 0,Y 149.373,Z 518.579,A -85,B 0,C 180,E1 -25160.918,E2 -25160.918} C_VEL
LIN {X 0,Y 155.45,Z 511.622,A -85,B 0,C 180,E1 -25164.46,E2 -25164.46} C_VEL
LIN {X 0,Y 160.9,Z 504.452,A -85,B 0,C 180,E1 -25167.219,E2 -25167.219} C_VEL
LIN {X 0,Y 167.173,Z 495.12,A -85,B 0,C 180,E1 -25169.891,E2 -25169.891} C_VEL
LIN {X 0,Y 172.88,Z 484.83,A -85,B 0,C 180,E1 -25172.144,E2 -25172.144} C_VEL
LIN {X 0,Y 177.971,Z 473.914,A -85,B 0,C 180,E1 -25173.938,E2 -25173.938} C_VEL
LIN {X 0,Y 182.311,Z 462.219,A -85,B 0,C 180,E1 -25175.397,E2 -25175.397} C_VEL
LIN {X 0,Y 185.651,Z 450.698,A -85,B 0,C 180,E1 -25176.441,E2 -25176.441} C_VEL
LIN {X 0,Y 188.411,Z 437.401,A -85,B 0,C 180,E1 -25177.289,E2 -25177.289} C_VEL
LIN {X 0,Y 190.015,Z 424.862,A -85,B 0,C 180,E1 -25177.769,E2 -25177.769} C_VEL
LIN {X 0,Y 191.15,Z 411.968,A -85,B 0,C 180,E1 -25178.145,E2 -25178.145} C_VEL
LIN {X 0,Y 191.049,Z 410.933,A -85,B 0,C 180,E1 -25178.275,E2 -25178.275} C_VEL
LIN {X 0,Y 186.794,Z 402.768,A -85,B 0,C 180,E1 -25181.328,E2 -25181.328} C_VEL
LIN {X 0,Y 183.326,Z 396.691,A -85,B 0,C 180,E1 -25184.167,E2 -25184.167} C_VEL
LIN {X 0,Y 180.729,Z 392.43,A -85,B 0,C 180,E1 -25186.574,E2 -25186.574} C_VEL
LIN {X 0,Y 178.86,Z 389.37,A -85,B 0,C 180,E1 -25188.529,E2 -25188.529} C_VEL
LIN {X 0,Y 176.727,Z 386.006,A -85,B 0,C 180,E1 -25191.067,E2 -25191.067} C_VEL
LIN {X 0,Y 174.416,Z 382.205,A -85,B 0,C 180,E1 -25194.509,E2 -25194.509} C_VEL
LIN {X 0,Y 171.956,Z 378.792,A -85,B 0,C 180,E1 -25199.744,E2 -25199.744} C_VEL
LIN {X 0,Y 171.468,Z 377.066,A -85,B 0,C 180,E1 -25201.734,E2 -25201.734} C_VEL
LIN {X 0,Y 170.925,Z 377.043,A -85,B 0,C 180,E1 -25210.527,E2 -25210.527} C_VEL
LIN {X 0,Y 171.403,Z 377.448,A -85,B 0,C 180,E1 -25212.743,E2 -25212.743} C_VEL
LIN {X 0,Y 173.257,Z 381.35,A -85,B 0,C 180,E1 -25218.066,E2 -25218.066} C_VEL
LIN {X 0,Y 174.334,Z 382.438,A -85,B 0,C 180,E1 -25219.959,E2 -25219.959} C_VEL
LIN {X 0,Y 177.45,Z 388.176,A -85,B 0,C 180,E1 -25224.509,E2 -25224.509} C_VEL
LIN {X 0,Y 180.036,Z 393.18,A -85,B 0,C 180,E1 -25227.474,E2 -25227.474} C_VEL
LIN {X 0,Y 183.406,Z 400.169,A -85,B 0,C 180,E1 -25230.763,E2 -25230.763} C_VEL
LIN {X 0,Y 187.154,Z 408.848,A -85,B 0,C 180,E1 -25233.944,E2 -25233.944} C_VEL
LIN {X 0,Y 190.604,Z 418.002,A -85,B 0,C 180,E1 -25236.557,E2 -25236.557} C_VEL
LIN {X 0,Y 188.43,Z 440.806,A -85,B 0,C 180,E1 -25237.321,E2 -25237.321} C_VEL
LIN {X 0,Y 185.956,Z 453.95,A -85,B 0,C 180,E1 -25237.994,E2 -25237.994} C_VEL
LIN {X 0,Y 182.634,Z 466.069,A -85,B 0,C 180,E1 -25238.919,E2 -25238.919} C_VEL
LIN {X 0,Y 178.182,Z 478.142,A -85,B 0,C 180,E1 -25240.17,E2 -25240.17} C_VEL
LIN {X 0,Y 173.086,Z 489.332,A -85,B 0,C 180,E1 -25241.753,E2 -25241.753} C_VEL
LIN {X 0,Y 167.598,Z 499.44,A -85,B 0,C 180,E1 -25243.674,E2 -25243.674} C_VEL
LIN {X 0,Y 161.801,Z 508.559,A -85,B 0,C 180,E1 -25245.981,E2 -25245.981} C_VEL
LIN {X 0,Y 155.277,Z 517.465,A -85,B 0,C 180,E1 -25248.988,E2 -25248.988} C_VEL
LIN {X 0,Y 149.166,Z 524.668,A -85,B 0,C 180,E1 -25252.235,E2 -25252.235} C_VEL
LIN {X 0,Y 143.709,Z 530.453,A -85,B 0,C 180,E1 -25255.784,E2 -25255.784} C_VEL
LIN {X 0,Y 139.109,Z 535.036,A -85,B 0,C 180,E1 -25259.66,E2 -25259.66} C_VEL
LIN {X 0,Y 134.978,Z 538.554,A -85,B 0,C 180,E1 -25263.737,E2 -25263.737} C_VEL
LIN {X 0,Y 131.614,Z 541.097,A -85,B 0,C 180,E1 -25268.056,E2 -25268.056} C_VEL
LIN {X 0,Y 129.793,Z 542.307,A -85,B 0,C 180,E1 -25271.047,E2 -25271.047} C_VEL
LIN {X 0,Y 127.484,Z 543.505,A -85,B 0,C 180,E1 -25277.266,E2 -25277.266} C_VEL
LIN {X 0,Y 126.545,Z 543.202,A -85,B 0,C 180,E1 -25283.628,E2 -25283.628} C_VEL
LIN {X 0,Y 126.545,Z 541.856,A -85,B 0,C 180,E1 -25288.573,E2 -25288.573} C_VEL
LIN {X 0,Y 126.535,Z 540.713,A -85,B 0,C 180,E1 -25291.236,E2 -25291.236} C_VEL
LIN {X 0,Y 126.564,Z 537.61,A -85,B 0,C 180,E1 -25296.381,E2 -25296.381} C_VEL
LIN {X 0,Y 127.265,Z 532.613,A -85,B 0,C 180,E1 -25302.132,E2 -25302.132} C_VEL
LIN {X 0,Y 128.785,Z 526.354,A -85,B 0,C 180,E1 -25307.471,E2 -25307.471} C_VEL
LIN {X 0,Y 131.057,Z 519.316,A -85,B 0,C 180,E1 -25312.052,E2 -25312.052} C_VEL
LIN {X 0,Y 131.944,Z 516.604,A -85,B 0,C 180,E1 -25313.531,E2 -25313.531} C_VEL
LIN {X 0,Y 132.175,Z 514.136,A -85,B 0,C 180,E1 -25314.886,E2 -25314.886} C_VEL
LIN {X 0,Y 130.879,Z 510.062,A -85,B 0,C 180,E1 -25317.167,E2 -25317.167} C_VEL
LIN {X 0,Y 129.693,Z 505.72,A -85,B 0,C 180,E1 -25319.389,E2 -25319.389} C_VEL
LIN {X 0,Y 130.078,Z 502.831,A -85,B 0,C 180,E1 -25320.592,E2 -25320.592} C_VEL
LIN {X 0,Y 133.076,Z 493.551,A -85,B 0,C 180,E1 -25323.683,E2 -25323.683} C_VEL
LIN {X 0,Y 135.911,Z 484.52,A -85,B 0,C 180,E1 -25326.035,E2 -25326.035} C_VEL
LIN {X 0,Y 138.971,Z 473.364,A -85,B 0,C 180,E1 -25328.285,E2 -25328.285} C_VEL
LIN {X 0,Y 141.803,Z 460.987,A -85,B 0,C 180,E1 -25330.118,E2 -25330.118} C_VEL
LIN {X 0,Y 143.969,Z 447.824,A -85,B 0,C 180,E1 -25331.463,E2 -25331.463} C_VEL
LIN {X 0,Y 145.278,Z 435.168,A -85,B 0,C 180,E1 -25332.283,E2 -25332.283} C_VEL
LIN {X 0,Y 147.59,Z 397.445,A -85,B 0,C 180,E1 -25333.926,E2 -25333.926} C_VEL
LIN {X 0,Y 146.6,Z 383.488,A -85,B 0,C 180,E1 -25335.084,E2 -25335.084} C_VEL
LIN {X 0,Y 142.195,Z 370.799,A -85,B 0,C 180,E1 -25337.338,E2 -25337.338} C_VEL
LIN {X 0,Y 137.933,Z 360.774,A -85,B 0,C 180,E1 -25339.578,E2 -25339.578} C_VEL
LIN {X 0,Y 135.404,Z 355.786,A -85,B 0,C 180,E1 -25340.945,E2 -25340.945} C_VEL
LIN {X 0,Y 130.501,Z 348.24,A -85,B 0,C 180,E1 -25343.672,E2 -25343.672} C_VEL
LIN {X 0,Y 128.05,Z 344.634,A -85,B 0,C 180,E1 -25345.148,E2 -25345.148} C_VEL
LIN {X 0,Y 125.862,Z 341.553,A -85,B 0,C 180,E1 -25346.535,E2 -25346.535} C_VEL
LIN {X 0,Y 125.126,Z 340.372,A -85,B 0,C 180,E1 -25347.035,E2 -25347.035} C_VEL
LIN {X 0,Y 122.966,Z 338.217,A -85,B 0,C 180,E1 -25348.444,E2 -25348.444} C_VEL
LIN {X 0,Y 121.96,Z 335.656,A -85,B 0,C 180,E1 -25349.283,E2 -25349.283} C_VEL
LIN {X 0,Y 121.919,Z 335.289,A -85,B 0,C 180,E1 -25349.446,E2 -25349.446} C_VEL
LIN {X 0,Y 121.948,Z 335.294,A -85,B 0,C 180,E1 -25352.544,E2 -25352.544} C_VEL
LIN {X 0,Y 122.017,Z 335.286,A -85,B 0,C 180,E1 -25357.169,E2 -25357.169} C_VEL
LIN {X 0,Y 122.073,Z 335.247,A -85,B 0,C 180,E1 -25363.269,E2 -25363.269} C_VEL
LIN {X 0,Y 122.296,Z 335.25,A -85,B 0,C 180,E1 -25367.691,E2 -25367.691} C_VEL
LIN {X 0,Y 122.421,Z 335.19,A -85,B 0,C 180,E1 -25373.406,E2 -25373.406} C_VEL
LIN {X 0,Y 123.048,Z 335.154,A -85,B 0,C 180,E1 -25379.999,E2 -25379.999} C_VEL
LIN {X 0,Y 122.408,Z 335.189,A -85,B 0,C 180,E1 -25386.916,E2 -25386.916} C_VEL
LIN {X 0,Y 122.297,Z 335.25,A -85,B 0,C 180,E1 -25392.31,E2 -25392.31} C_VEL
LIN {X 0,Y 122.084,Z 335.267,A -85,B 0,C 180,E1 -25396.728,E2 -25396.728} C_VEL
LIN {X 0,Y 122.035,Z 335.272,A -85,B 0,C 180,E1 -25402.851,E2 -25402.851} C_VEL
LIN {X 0,Y 121.948,Z 335.285,A -85,B 0,C 180,E1 -25407.454,E2 -25407.454} C_VEL
LIN {X 0,Y 121.907,Z 335.295,A -85,B 0,C 180,E1 -25411.255,E2 -25411.255} C_VEL
LIN {X 0,Y 121.891,Z 335.291,A -85,B 0,C 180,E1 -25416.168,E2 -25416.168} C_VEL
LIN {X 0,Y 121.875,Z 335.291,A -85,B 0,C 180,E1 -25421.433,E2 -25421.433} C_VEL
LIN {X 0,Y 121.844,Z 335.296,A -85,B 0,C 180,E1 -25426.192,E2 -25426.192} C_VEL
LIN {X 0,Y 122.678,Z 337.903,A -85,B 0,C 180,E1 -25426.969,E2 -25426.969} C_VEL
LIN {X 0,Y 124.631,Z 340.09,A -85,B 0,C 180,E1 -25428.281,E2 -25428.281} C_VEL
LIN {X 0,Y 125.559,Z 341.012,A -85,B 0,C 180,E1 -25428.868,E2 -25428.868} C_VEL
LIN {X 0,Y 127.684,Z 344.267,A -85,B 0,C 180,E1 -25430.252,E2 -25430.252} C_VEL
LIN {X 0,Y 128.857,Z 345.751,A -85,B 0,C 180,E1 -25430.955,E2 -25430.955} C_VEL
LIN {X 0,Y 134.346,Z 353.894,A -85,B 0,C 180,E1 -25434.076,E2 -25434.076} C_VEL
LIN {X 0,Y 141.124,Z 365.6,A -85,B 0,C 180,E1 -25437.543,E2 -25437.543} C_VEL
LIN {X 0,Y 146.809,Z 377.417,A -85,B 0,C 180,E1 -25440.208,E2 -25440.208} C_VEL
LIN {X 0,Y 148.551,Z 381.404,A -85,B 0,C 180,E1 -25440.988,E2 -25440.988} C_VEL
LIN {X 0,Y 145.097,Z 431.553,A -85,B 0,C 180,E1 -25443.143,E2 -25443.143} C_VEL
LIN {X 0,Y 143.376,Z 444.824,A -85,B 0,C 180,E1 -25444.208,E2 -25444.208} C_VEL
LIN {X 0,Y 141.3,Z 457.222,A -85,B 0,C 180,E1 -25445.769,E2 -25445.769} C_VEL
LIN {X 0,Y 138.671,Z 468.392,A -85,B 0,C 180,E1 -25447.655,E2 -25447.655} C_VEL
LIN {X 0,Y 135.857,Z 478.689,A -85,B 0,C 180,E1 -25449.953,E2 -25449.953} C_VEL
LIN {X 0,Y 133.004,Z 487.968,A -85,B 0,C 180,E1 -25452.593,E2 -25452.593} C_VEL
LIN {X 0,Y 129.883,Z 497.168,A -85,B 0,C 180,E1 -25455.902,E2 -25455.902} C_VEL
LIN {X 0,Y 126.903,Z 505.351,A -85,B 0,C 180,E1 -25459.626,E2 -25459.626} C_VEL
LIN {X 0,Y 123.992,Z 513.379,A -85,B 0,C 180,E1 -25464.303,E2 -25464.303} C_VEL
LIN {X 0,Y 122.17,Z 518.799,A -85,B 0,C 180,E1 -25468.347,E2 -25468.347} C_VEL
LIN {X 0,Y 120.613,Z 524.113,A -85,B 0,C 180,E1 -25473.335,E2 -25473.335} C_VEL
LIN {X 0,Y 119.495,Z 528.27,A -85,B 0,C 180,E1 -25478.45,E2 -25478.45} C_VEL
LIN {X 0,Y 118.995,Z 531.357,A -85,B 0,C 180,E1 -25483.66,E2 -25483.66} C_VEL
LIN {X 0,Y 119.369,Z 533.639,A -85,B 0,C 180,E1 -25489.608,E2 -25489.608} C_VEL
LIN {X 0,Y 120.176,Z 534.557,A -85,B 0,C 180,E1 -25494.159,E2 -25494.159} C_VEL
LIN {X 0,Y 121.261,Z 534.785,A -85,B 0,C 180,E1 -25497.618,E2 -25497.618} C_VEL
LIN {X 0,Y 122.694,Z 534.56,A -85,B 0,C 180,E1 -25501.026,E2 -25501.026} C_VEL
LIN {X 0,Y 124.492,Z 533.928,A -85,B 0,C 180,E1 -25504.364,E2 -25504.364} C_VEL
LIN {X 0,Y 128.748,Z 531.664,A -85,B 0,C 180,E1 -25510.163,E2 -25510.163} C_VEL
LIN {X 0,Y 133.691,Z 528.16,A -85,B 0,C 180,E1 -25515.202,E2 -25515.202} C_VEL
LIN {X 0,Y 138.915,Z 523.833,A -85,B 0,C 180,E1 -25519.358,E2 -25519.358} C_VEL
LIN {X 0,Y 144.794,Z 518.216,A -85,B 0,C 180,E1 -25523.206,E2 -25523.206} C_VEL
LIN {X 0,Y 151.228,Z 511.115,A -85,B 0,C 180,E1 -25526.765,E2 -25526.765} C_VEL
LIN {X 0,Y 157.019,Z 503.779,A -85,B 0,C 180,E1 -25529.489,E2 -25529.489} C_VEL
LIN {X 0,Y 163.768,Z 493.817,A -85,B 0,C 180,E1 -25532.233,E2 -25532.233} C_VEL
LIN {X 0,Y 169.542,Z 483.622,A -85,B 0,C 180,E1 -25534.36,E2 -25534.36} C_VEL
LIN {X 0,Y 174.534,Z 473.039,A -85,B 0,C 180,E1 -25536.018,E2 -25536.018} C_VEL
LIN {X 0,Y 179.192,Z 460.387,A -85,B 0,C 180,E1 -25537.528,E2 -25537.528} C_VEL
LIN {X 0,Y 182.644,Z 448.409,A -85,B 0,C 180,E1 -25538.517,E2 -25538.517} C_VEL
LIN {X 0,Y 185.114,Z 436.016,A -85,B 0,C 180,E1 -25539.248,E2 -25539.248} C_VEL
LIN {X 0,Y 186.915,Z 420.473,A -85,B 0,C 180,E1 -25539.779,E2 -25539.779} C_VEL
LIN {X 0,Y 187.45,Z 414.684,A -85,B 0,C 180,E1 -25539.943,E2 -25539.943} C_VEL
LIN {X 0,Y 183.118,Z 406.108,A -85,B 0,C 180,E1 -25543.41,E2 -25543.41} C_VEL
LIN {X 0,Y 179.199,Z 399.298,A -85,B 0,C 180,E1 -25547.077,E2 -25547.077} C_VEL
LIN {X 0,Y 177.072,Z 395.688,A -85,B 0,C 180,E1 -25549.423,E2 -25549.423} C_VEL
LIN {X 0,Y 175.227,Z 392.636,A -85,B 0,C 180,E1 -25551.766,E2 -25551.766} C_VEL
LIN {X 0,Y 173.016,Z 388.744,A -85,B 0,C 180,E1 -25555.341,E2 -25555.341} C_VEL
LIN {X 0,Y 170.999,Z 385.962,A -85,B 0,C 180,E1 -25559.872,E2 -25559.872} C_VEL
LIN {X 0,Y 170.542,Z 384.222,A -85,B 0,C 180,E1 -25561.82,E2 -25561.82} C_VEL
LIN {X 0,Y 169.902,Z 383.982,A -85,B 0,C 180,E1 -25569.525,E2 -25569.525} C_VEL
LIN {X 0,Y 170.43,Z 384.517,A -85,B 0,C 180,E1 -25572.449,E2 -25572.449} C_VEL
LIN {X 0,Y 172.105,Z 388.196,A -85,B 0,C 180,E1 -25577.576,E2 -25577.576} C_VEL
LIN {X 0,Y 173.13,Z 389.376,A -85,B 0,C 180,E1 -25579.498,E2 -25579.498} C_VEL
LIN {X 0,Y 175.797,Z 394.607,A -85,B 0,C 180,E1 -25583.673,E2 -25583.673} C_VEL
LIN {X 0,Y 178.04,Z 399.204,A -85,B 0,C 180,E1 -25586.444,E2 -25586.444} C_VEL
LIN {X 0,Y 181.159,Z 406.046,A -85,B 0,C 180,E1 -25589.724,E2 -25589.724} C_VEL
LIN {X 0,Y 184.426,Z 414.06,A -85,B 0,C 180,E1 -25592.718,E2 -25592.718} C_VEL
LIN {X 0,Y 186.912,Z 421.004,A -85,B 0,C 180,E1 -25594.804,E2 -25594.804} C_VEL
LIN {X 0,Y 184.847,Z 440.833,A -85,B 0,C 180,E1 -25595.444,E2 -25595.444} C_VEL
LIN {X 0,Y 182.351,Z 453.655,A -85,B 0,C 180,E1 -25596.09,E2 -25596.09} C_VEL
LIN {X 0,Y 179.016,Z 465.526,A -85,B 0,C 180,E1 -25596.973,E2 -25596.973} C_VEL
LIN {X 0,Y 174.401,Z 477.732,A -85,B 0,C 180,E1 -25598.211,E2 -25598.211} C_VEL
LIN {X 0,Y 169.102,Z 488.956,A -85,B 0,C 180,E1 -25599.754,E2 -25599.754} C_VEL
LIN {X 0,Y 163.396,Z 499.09,A -85,B 0,C 180,E1 -25601.646,E2 -25601.646} C_VEL
LIN {X 0,Y 156.791,Z 509.033,A -85,B 0,C 180,E1 -25604.184,E2 -25604.184} C_VEL
LIN {X 0,Y 149.996,Z 517.816,A -85,B 0,C 180,E1 -25607.21,E2 -25607.21} C_VEL
LIN {X 0,Y 143.633,Z 524.891,A -85,B 0,C 180,E1 -25610.505,E2 -25610.505} C_VEL
LIN {X 0,Y 137.878,Z 530.564,A -85,B 0,C 180,E1 -25614.119,E2 -25614.119} C_VEL
LIN {X 0,Y 133.002,Z 535.064,A -85,B 0,C 180,E1 -25618.108,E2 -25618.108} C_VEL
LIN {X 0,Y 127.358,Z 539.426,A -85,B 0,C 180,E1 -25623.808,E2 -25623.808} C_VEL
LIN {X 0,Y 125.038,Z 540.996,A -85,B 0,C 180,E1 -25626.836,E2 -25626.836} C_VEL
LIN {X 0,Y 123.072,Z 542.136,A -85,B 0,C 180,E1 -25629.968,E2 -25629.968} C_VEL
LIN {X 0,Y 120.544,Z 543.257,A -85,B 0,C 180,E1 -25636.519,E2 -25636.519} C_VEL
LIN {X 0,Y 119.47,Z 542.867,A -85,B 0,C 180,E1 -25643.248,E2 -25643.248} C_VEL
LIN {X 0,Y 119.489,Z 541.169,A -85,B 0,C 180,E1 -25649.218,E2 -25649.218} C_VEL
LIN {X 0,Y 119.403,Z 538.172,A -85,B 0,C 180,E1 -25655.07,E2 -25655.07} C_VEL
LIN {X 0,Y 119.838,Z 534.451,A -85,B 0,C 180,E1 -25660.138,E2 -25660.138} C_VEL
LIN {X 0,Y 120.848,Z 529.565,A -85,B 0,C 180,E1 -25665.176,E2 -25665.176} C_VEL
LIN {X 0,Y 122.775,Z 523.389,A -85,B 0,C 180,E1 -25670.093,E2 -25670.093} C_VEL
LIN {X 0,Y 125.454,Z 515.68,A -85,B 0,C 180,E1 -25674.849,E2 -25674.849} C_VEL
LIN {X 0,Y 127.656,Z 509.037,A -85,B 0,C 180,E1 -25678.112,E2 -25678.112} C_VEL
LIN {X 0,Y 130.078,Z 502.831,A -85,B 0,C 180,E1 -25680.592,E2 -25680.592} C_VEL
LIN {X 0,Y 130.46,Z 499.906,A -85,B 0,C 180,E1 -25681.773,E2 -25681.773} C_VEL
LIN {X 0,Y 129.343,Z 495.211,A -85,B 0,C 180,E1 -25683.865,E2 -25683.865} C_VEL
LIN {X 0,Y 128.34,Z 490.313,A -85,B 0,C 180,E1 -25685.903,E2 -25685.903} C_VEL
LIN {X 0,Y 128.825,Z 487.057,A -85,B 0,C 180,E1 -25686.906,E2 -25686.906} C_VEL
LIN {X 0,Y 132.082,Z 476.771,A -85,B 0,C 180,E1 -25689.193,E2 -25689.193} C_VEL
LIN {X 0,Y 134.923,Z 465.483,A -85,B 0,C 180,E1 -25691.124,E2 -25691.124} C_VEL
LIN {X 0,Y 137.481,Z 452.323,A -85,B 0,C 180,E1 -25692.715,E2 -25692.715} C_VEL
LIN {X 0,Y 139.178,Z 439.673,A -85,B 0,C 180,E1 -25693.724,E2 -25693.724} C_VEL
LIN {X 0,Y 141.979,Z 398.31,A -85,B 0,C 180,E1 -25695.607,E2 -25695.607} C_VEL
LIN {X 0,Y 141.193,Z 385.802,A -85,B 0,C 180,E1 -25696.687,E2 -25696.687} C_VEL
LIN {X 0,Y 136.87,Z 373.23,A -85,B 0,C 180,E1 -25699.103,E2 -25699.103} C_VEL
LIN {X 0,Y 133.216,Z 364.486,A -85,B 0,C 180,E1 -25701.208,E2 -25701.208} C_VEL
LIN {X 0,Y 131.261,Z 360.538,A -85,B 0,C 180,E1 -25702.358,E2 -25702.358} C_VEL
LIN {X 0,Y 126.672,Z 353.362,A -85,B 0,C 180,E1 -25705.098,E2 -25705.098} C_VEL
LIN {X 0,Y 124.016,Z 349.472,A -85,B 0,C 180,E1 -25706.823,E2 -25706.823} C_VEL
LIN {X 0,Y 121.701,Z 346.082,A -85,B 0,C 180,E1 -25708.442,E2 -25708.442} C_VEL
LIN {X 0,Y 119.302,Z 343.09,A -85,B 0,C 180,E1 -25710.201,E2 -25710.201} C_VEL
LIN {X 0,Y 118.392,Z 341.454,A -85,B 0,C 180,E1 -25710.958,E2 -25710.958} C_VEL
LIN {X 0,Y 116.108,Z 339.349,A -85,B 0,C 180,E1 -25712.757,E2 -25712.757} C_VEL
